LIN {X 0,Y 263.736,Z 330.131,A -85,B 0,C 180,E1 -17998.473,E2 -17998.473} C_VEL
LIN {X 0,Y 263.74,Z 330.122,A -85,B 0,C 180,E1 -18001.527,E2 -18001.527} C_VEL
LIN {X 0,Y 263.538,Z 330.145,A -85,B 0,C 180,E1 -18007.662,E2 -18007.662} C_VEL
LIN {X 0,Y 263.345,Z 330.181,A -85,B 0,C 180,E1 -18010.766,E2 -18010.766} C_VEL
LIN {X 0,Y 263.289,Z 330.157,A -85,B 0,C 180,E1 -18015.481,E2 -18015.481} C_VEL
LIN {X 0,Y 263.209,Z 330.198,A -85,B 0,C 180,E1 -18020.311,E2 -18020.311} C_VEL
LIN {X 0,Y 263.167,Z 330.188,A -85,B 0,C 180,E1 -18025.295,E2 -18025.295} C_VEL
LIN {X 0,Y 263.133,Z 330.206,A -85,B 0,C 180,E1 -18028.735,E2 -18028.735} C_VEL
LIN {X 0,Y 263.128,Z 330.196,A -85,B 0,C 180,E1 -18032.288,E2 -18032.288} C_VEL
LIN {X 0,Y 263.153,Z 330.198,A -85,B 0,C 180,E1 -18035.983,E2 -18035.983} C_VEL
LIN {X 0,Y 263.071,Z 330.217,A -85,B 0,C 180,E1 -18039.878,E2 -18039.878} C_VEL
LIN {X 0,Y 263.075,Z 330.212,A -85,B 0,C 180,E1 -18043.993,E2 -18043.993} C_VEL
LIN {X 0,Y 263.079,Z 330.215,A -85,B 0,C 180,E1 -18048.417,E2 -18048.417} C_VEL
LIN {X 0,Y 263.155,Z 330.203,A -85,B 0,C 180,E1 -18052.102,E2 -18052.102} C_VEL
LIN {X 0,Y 263.202,Z 330.409,A -85,B 0,C 180,E1 -18055.314,E2 -18055.314} C_VEL
LIN {X 0,Y 265.444,Z 340.558,A -85,B 0,C 180,E1 -18059.358,E2 -18059.358} C_VEL
LIN {X 0,Y 266.018,Z 343.587,A -85,B 0,C 180,E1 -18060.39,E2 -18060.39} C_VEL
LIN {X 0,Y 270.223,Z 354.313,A -85,B 0,C 180,E1 -18061.21,E2 -18061.21} C_VEL
LIN {X 0,Y 273.348,Z 362.999,A -85,B 0,C 180,E1 -18061.777,E2 -18061.777} C_VEL
LIN {X 0,Y 277.181,Z 387.27,A -85,B 0,C 180,E1 -18062.845,E2 -18062.845} C_VEL
LIN {X 0,Y 275.215,Z 449.746,A -85,B 0,C 180,E1 -18064.524,E2 -18064.524} C_VEL
LIN {X 0,Y 274.623,Z 459.446,A -85,B 0,C 180,E1 -18064.921,E2 -18064.921} C_VEL
LIN {X 0,Y 273.731,Z 469.978,A -85,B 0,C 180,E1 -18065.543,E2 -18065.543} C_VEL
LIN {X 0,Y 272.657,Z 479.225,A -85,B 0,C 180,E1 -18066.25,E2 -18066.25} C_VEL
LIN {X 0,Y 271.281,Z 490.013,A -85,B 0,C 180,E1 -18067.334,E2 -18067.334} C_VEL
LIN {X 0,Y 269.73,Z 500.089,A -85,B 0,C 180,E1 -18068.606,E2 -18068.606} C_VEL
LIN {X 0,Y 268.138,Z 509.514,A -85,B 0,C 180,E1 -18070.078,E2 -18070.078} C_VEL
LIN {X 0,Y 266.815,Z 517.421,A -85,B 0,C 180,E1 -18071.573,E2 -18071.573} C_VEL
LIN {X 0,Y 265.298,Z 525.618,A -85,B 0,C 180,E1 -18073.454,E2 -18073.454} C_VEL
LIN {X 0,Y 264.028,Z 532.435,A -85,B 0,C 180,E1 -18075.352,E2 -18075.352} C_VEL
LIN {X 0,Y 263.156,Z 537.135,A -85,B 0,C 180,E1 -18076.879,E2 -18076.879} C_VEL
LIN {X 0,Y 262.228,Z 542.864,A -85,B 0,C 180,E1 -18079.187,E2 -18079.187} C_VEL
LIN {X 0,Y 261.569,Z 547.363,A -85,B 0,C 180,E1 -18081.502,E2 -18081.502} C_VEL
LIN {X 0,Y 261.166,Z 550.77,A -85,B 0,C 180,E1 -18083.821,E2 -18083.821} C_VEL
LIN {X 0,Y 261.007,Z 553.667,A -85,B 0,C 180,E1 -18086.913,E2 -18086.913} C_VEL
LIN {X 0,Y 261.032,Z 554.618,A -85,B 0,C 180,E1 -18088.457,E2 -18088.457} C_VEL
LIN {X 0,Y 261.033,Z 555.058,A -85,B 0,C 180,E1 -18091.543,E2 -18091.543} C_VEL
LIN {X 0,Y 261.013,Z 554.722,A -85,B 0,C 180,E1 -18093.087,E2 -18093.087} C_VEL
LIN {X 0,Y 261.231,Z 552.837,A -85,B 0,C 180,E1 -18096.178,E2 -18096.178} C_VEL
LIN {X 0,Y 261.634,Z 550.327,A -85,B 0,C 180,E1 -18098.496,E2 -18098.496} C_VEL
LIN {X 0,Y 262.351,Z 546.813,A -85,B 0,C 180,E1 -18100.808,E2 -18100.808} C_VEL
LIN {X 0,Y 263.39,Z 542.211,A -85,B 0,C 180,E1 -18103.109,E2 -18103.109} C_VEL
LIN {X 0,Y 264.878,Z 536.377,A -85,B 0,C 180,E1 -18105.386,E2 -18105.386} C_VEL
LIN {X 0,Y 266.728,Z 529.069,A -85,B 0,C 180,E1 -18107.639,E2 -18107.639} C_VEL
LIN {X 0,Y 268.25,Z 522.147,A -85,B 0,C 180,E1 -18109.409,E2 -18109.409} C_VEL
LIN {X 0,Y 270.195,Z 513.761,A -85,B 0,C 180,E1 -18111.155,E2 -18111.155} C_VEL
LIN {X 0,Y 272.29,Z 504.136,A -85,B 0,C 180,E1 -18112.778,E2 -18112.778} C_VEL
LIN {X 0,Y 274.149,Z 495.111,A -85,B 0,C 180,E1 -18114.014,E2 -18114.014} C_VEL
LIN {X 0,Y 275.782,Z 485.768,A -85,B 0,C 180,E1 -18115.066,E2 -18115.066} C_VEL
LIN {X 0,Y 277.322,Z 475.015,A -85,B 0,C 180,E1 -18116.023,E2 -18116.023} C_VEL
LIN {X 0,Y 278.606,Z 464.155,A -85,B 0,C 180,E1 -18116.751,E2 -18116.751} C_VEL
LIN {X 0,Y 279.679,Z 453.063,A -85,B 0,C 180,E1 -18117.266,E2 -18117.266} C_VEL
LIN {X 0,Y 280.37,Z 435.148,A -85,B 0,C 180,E1 -18117.818,E2 -18117.818} C_VEL
LIN {X 0,Y 282.056,Z 388.472,A -85,B 0,C 180,E1 -18119.049,E2 -18119.049} C_VEL
LIN {X 0,Y 279.053,Z 370.079,A -85,B 0,C 180,E1 -18120.029,E2 -18120.029} C_VEL
LIN {X 0,Y 272.265,Z 354.512,A -85,B 0,C 180,E1 -18121.501,E2 -18121.501} C_VEL
LIN {X 0,Y 267.461,Z 345.107,A -85,B 0,C 180,E1 -18122.57,E2 -18122.57} C_VEL
LIN {X 0,Y 266.322,Z 342.4,A -85,B 0,C 180,E1 -18122.941,E2 -18122.941} C_VEL
LIN {X 0,Y 264.141,Z 333.763,A -85,B 0,C 180,E1 -18126.565,E2 -18126.565} C_VEL
LIN {X 0,Y 263.175,Z 330.249,A -85,B 0,C 180,E1 -18128.281,E2 -18128.281} C_VEL
LIN {X 0,Y 263.122,Z 330.208,A -85,B 0,C 180,E1 -18131.894,E2 -18131.894} C_VEL
LIN {X 0,Y 263.103,Z 330.208,A -85,B 0,C 180,E1 -18136.155,E2 -18136.155} C_VEL
LIN {X 0,Y 263.104,Z 330.212,A -85,B 0,C 180,E1 -18140.128,E2 -18140.128} C_VEL
LIN {X 0,Y 263.161,Z 330.2,A -85,B 0,C 180,E1 -18144.018,E2 -18144.018} C_VEL
LIN {X 0,Y 263.132,Z 330.203,A -85,B 0,C 180,E1 -18147.712,E2 -18147.712} C_VEL
LIN {X 0,Y 263.198,Z 330.194,A -85,B 0,C 180,E1 -18151.785,E2 -18151.785} C_VEL
LIN {X 0,Y 263.226,Z 330.195,A -85,B 0,C 180,E1 -18155.201,E2 -18155.201} C_VEL
LIN {X 0,Y 263.264,Z 330.19,A -85,B 0,C 180,E1 -18159.694,E2 -18159.694} C_VEL
LIN {X 0,Y 263.351,Z 330.179,A -85,B 0,C 180,E1 -18164.522,E2 -18164.522} C_VEL
LIN {X 0,Y 263.375,Z 330.178,A -85,B 0,C 180,E1 -18169.235,E2 -18169.235} C_VEL
LIN {X 0,Y 263.575,Z 330.146,A -85,B 0,C 180,E1 -18172.339,E2 -18172.339} C_VEL
LIN {X 0,Y 263.753,Z 330.131,A -85,B 0,C 180,E1 -18178.473,E2 -18178.473} C_VEL
LIN {X 0,Y 263.753,Z 330.125,A -85,B 0,C 180,E1 -18181.527,E2 -18181.527} C_VEL
LIN {X 0,Y 263.574,Z 330.15,A -85,B 0,C 180,E1 -18187.662,E2 -18187.662} C_VEL
LIN {X 0,Y 263.376,Z 330.178,A -85,B 0,C 180,E1 -18190.766,E2 -18190.766} C_VEL
LIN {X 0,Y 263.352,Z 330.176,A -85,B 0,C 180,E1 -18195.478,E2 -18195.478} C_VEL
LIN {X 0,Y 263.263,Z 330.192,A -85,B 0,C 180,E1 -18200.307,E2 -18200.307} C_VEL
LIN {X 0,Y 263.186,Z 330.202,A -85,B 0,C 180,E1 -18205.294,E2 -18205.294} C_VEL
LIN {X 0,Y 263.164,Z 330.203,A -85,B 0,C 180,E1 -18209.828,E2 -18209.828} C_VEL
LIN {X 0,Y 263.23,Z 330.519,A -85,B 0,C 180,E1 -18210.262,E2 -18210.262} C_VEL
LIN {X 0,Y 264.944,Z 336.603,A -85,B 0,C 180,E1 -18212.886,E2 -18212.886} C_VEL
LIN {X 0,Y 267.825,Z 342.072,A -85,B 0,C 180,E1 -18213.63,E2 -18213.63} C_VEL
LIN {X 0,Y 274.766,Z 355.657,A -85,B 0,C 180,E1 -18215.15,E2 -18215.15} C_VEL
LIN {X 0,Y 281.344,Z 371.108,A -85,B 0,C 180,E1 -18216.558,E2 -18216.558} C_VEL
LIN {X 0,Y 282.522,Z 377.532,A -85,B 0,C 180,E1 -18216.915,E2 -18216.915} C_VEL
LIN {X 0,Y 279.879,Z 443.081,A -85,B 0,C 180,E1 -18218.66,E2 -18218.66} C_VEL
LIN {X 0,Y 279.168,Z 453.092,A -85,B 0,C 180,E1 -18219.075,E2 -18219.075} C_VEL
LIN {X 0,Y 278.267,Z 462.472,A -85,B 0,C 180,E1 -18219.618,E2 -18219.618} C_VEL
LIN {X 0,Y 276.999,Z 472.966,A -85,B 0,C 180,E1 -18220.434,E2 -18220.434} C_VEL
LIN {X 0,Y 275.434,Z 482.994,A -85,B 0,C 180,E1 -18221.423,E2 -18221.423} C_VEL
LIN {X 0,Y 273.661,Z 493.048,A -85,B 0,C 180,E1 -18222.682,E2 -18222.682} C_VEL
LIN {X 0,Y 271.796,Z 502.27,A -85,B 0,C 180,E1 -18224.104,E2 -18224.104} C_VEL
LIN {X 0,Y 269.717,Z 511.296,A -85,B 0,C 180,E1 -18225.812,E2 -18225.812} C_VEL
LIN {X 0,Y 267.874,Z 518.886,A -85,B 0,C 180,E1 -18227.565,E2 -18227.565} C_VEL
LIN {X 0,Y 266.451,Z 524.682,A -85,B 0,C 180,E1 -18229.155,E2 -18229.155} C_VEL
LIN {X 0,Y 264.768,Z 531.329,A -85,B 0,C 180,E1 -18231.407,E2 -18231.407} C_VEL
LIN {X 0,Y 263.723,Z 535.462,A -85,B 0,C 180,E1 -18233.08,E2 -18233.08} C_VEL
LIN {X 0,Y 262.444,Z 540.564,A -85,B 0,C 180,E1 -18235.781,E2 -18235.781} C_VEL
LIN {X 0,Y 261.865,Z 543.167,A -85,B 0,C 180,E1 -18237.536,E2 -18237.536} C_VEL
LIN {X 0,Y 261.377,Z 545.131,A -85,B 0,C 180,E1 -18239.365,E2 -18239.365} C_VEL
LIN {X 0,Y 260.81,Z 547.438,A -85,B 0,C 180,E1 -18242.736,E2 -18242.736} C_VEL
LIN {X 0,Y 260.66,Z 547.783,A -85,B 0,C 180,E1 -18244.444,E2 -18244.444} C_VEL
LIN {X 0,Y 260.664,Z 547.185,A -85,B 0,C 180,E1 -18247.823,E2 -18247.823} C_VEL
LIN {X 0,Y 260.965,Z 545.286,A -85,B 0,C 180,E1 -18250.49,E2 -18250.49} C_VEL
LIN {X 0,Y 261.376,Z 542.668,A -85,B 0,C 180,E1 -18252.796,E2 -18252.796} C_VEL
LIN {X 0,Y 261.913,Z 539.194,A -85,B 0,C 180,E1 -18255.017,E2 -18255.017} C_VEL
LIN {X 0,Y 262.505,Z 535.554,A -85,B 0,C 180,E1 -18256.846,E2 -18256.846} C_VEL
LIN {X 0,Y 263.528,Z 529.579,A -85,B 0,C 180,E1 -18259.241,E2 -18259.241} C_VEL
LIN {X 0,Y 264.959,Z 521.962,A -85,B 0,C 180,E1 -18261.612,E2 -18261.612} C_VEL
LIN {X 0,Y 266.44,Z 514.196,A -85,B 0,C 180,E1 -18263.564,E2 -18263.564} C_VEL
LIN {X 0,Y 267.763,Z 506.654,A -85,B 0,C 180,E1 -18265.145,E2 -18265.145} C_VEL
LIN {X 0,Y 269.281,Z 498.066,A -85,B 0,C 180,E1 -18266.634,E2 -18266.634} C_VEL
LIN {X 0,Y 270.742,Z 488.817,A -85,B 0,C 180,E1 -18267.955,E2 -18267.955} C_VEL
LIN {X 0,Y 272.075,Z 479.203,A -85,B 0,C 180,E1 -18269.075,E2 -18269.075} C_VEL
LIN {X 0,Y 273.277,Z 469.269,A -85,B 0,C 180,E1 -18270,E2 -18270} C_VEL
LIN {X 0,Y 274.319,Z 457.387,A -85,B 0,C 180,E1 -18270.836,E2 -18270.836} C_VEL
LIN {X 0,Y 275.192,Z 445.994,A -85,B 0,C 180,E1 -18271.385,E2 -18271.385} C_VEL
LIN {X 0,Y 275.864,Z 428.906,A -85,B 0,C 180,E1 -18271.899,E2 -18271.899} C_VEL
LIN {X 0,Y 277.459,Z 374.822,A -85,B 0,C 180,E1 -18273.325,E2 -18273.325} C_VEL
LIN {X 0,Y 275.15,Z 362.729,A -85,B 0,C 180,E1 -18273.899,E2 -18273.899} C_VEL
LIN {X 0,Y 269.038,Z 346.952,A -85,B 0,C 180,E1 -18274.974,E2 -18274.974} C_VEL
LIN {X 0,Y 264.977,Z 337.261,A -85,B 0,C 180,E1 -18275.747,E2 -18275.747} C_VEL
LIN {X 0,Y 264.714,Z 335.941,A -85,B 0,C 180,E1 -18276.096,E2 -18276.096} C_VEL
LIN {X 0,Y 263.505,Z 330.211,A -85,B 0,C 180,E1 -18278.548,E2 -18278.548} C_VEL
LIN {X 0,Y 263.324,Z 330.174,A -85,B 0,C 180,E1 -18282.329,E2 -18282.329} C_VEL
LIN {X 0,Y 263.349,Z 330.177,A -85,B 0,C 180,E1 -18286.109,E2 -18286.109} C_VEL
LIN {X 0,Y 263.216,Z 330.199,A -85,B 0,C 180,E1 -18290.849,E2 -18290.849} C_VEL
LIN {X 0,Y 263.195,Z 330.201,A -85,B 0,C 180,E1 -18295.293,E2 -18295.293} C_VEL
LIN {X 0,Y 263.168,Z 330.189,A -85,B 0,C 180,E1 -18298.731,E2 -18298.731} C_VEL
LIN {X 0,Y 263.135,Z 330.204,A -85,B 0,C 180,E1 -18302.288,E2 -18302.288} C_VEL
LIN {X 0,Y 263.189,Z 330.191,A -85,B 0,C 180,E1 -18305.978,E2 -18305.978} C_VEL
LIN {X 0,Y 263.117,Z 330.198,A -85,B 0,C 180,E1 -18309.871,E2 -18309.871} C_VEL
LIN {X 0,Y 263.13,Z 330.199,A -85,B 0,C 180,E1 -18313.983,E2 -18313.983} C_VEL
LIN {X 0,Y 263.127,Z 330.193,A -85,B 0,C 180,E1 -18318.406,E2 -18318.406} C_VEL
LIN {X 0,Y 263.16,Z 330.185,A -85,B 0,C 180,E1 -18322.103,E2 -18322.103} C_VEL
LIN {X 0,Y 263.153,Z 330.202,A -85,B 0,C 180,E1 -18325.885,E2 -18325.885} C_VEL
LIN {X 0,Y 263.128,Z 330.174,A -85,B 0,C 180,E1 -18329.504,E2 -18329.504} C_VEL
LIN {X 0,Y 263.151,Z 330.19,A -85,B 0,C 180,E1 -18332.998,E2 -18332.998} C_VEL
LIN {X 0,Y 263.152,Z 330.206,A -85,B 0,C 180,E1 -18336.384,E2 -18336.384} C_VEL
LIN {X 0,Y 263.24,Z 330.172,A -85,B 0,C 180,E1 -18339.691,E2 -18339.691} C_VEL
LIN {X 0,Y 263.317,Z 330.165,A -85,B 0,C 180,E1 -18344.52,E2 -18344.52} C_VEL
LIN {X 0,Y 263.355,Z 330.176,A -85,B 0,C 180,E1 -18349.233,E2 -18349.233} C_VEL
LIN {X 0,Y 263.528,Z 330.124,A -85,B 0,C 180,E1 -18352.337,E2 -18352.337} C_VEL
LIN {X 0,Y 263.478,Z 330.122,A -85,B 0,C 180,E1 -18353.306,E2 -18353.306} C_VEL
LIN {X 0,Y 262.843,Z 330.206,A -85,B 0,C 180,E1 -18354.581,E2 -18354.581} C_VEL
LIN {X 0,Y 260.134,Z 330.568,A -85,B 0,C 180,E1 -18356.665,E2 -18356.665} C_VEL
LIN {X 0,Y 257.028,Z 330.971,A -85,B 0,C 180,E1 -18359.227,E2 -18359.227} C_VEL
LIN {X 0,Y 256.696,Z 331.007,A -85,B 0,C 180,E1 -18360.112,E2 -18360.112} C_VEL
LIN {X 0,Y 256.702,Z 330.999,A -85,B 0,C 180,E1 -18361.568,E2 -18361.568} C_VEL
LIN {X 0,Y 256.464,Z 331.01,A -85,B 0,C 180,E1 -18366.293,E2 -18366.293} C_VEL
LIN {X 0,Y 256.428,Z 331.044,A -85,B 0,C 180,E1 -18369.464,E2 -18369.464} C_VEL
LIN {X 0,Y 256.207,Z 331.04,A -85,B 0,C 180,E1 -18374.292,E2 -18374.292} C_VEL
LIN {X 0,Y 256.149,Z 331.066,A -85,B 0,C 180,E1 -18377.566,E2 -18377.566} C_VEL
LIN {X 0,Y 256.122,Z 331.076,A -85,B 0,C 180,E1 -18381.098,E2 -18381.098} C_VEL
LIN {X 0,Y 256.133,Z 331.061,A -85,B 0,C 180,E1 -18385.111,E2 -18385.111} C_VEL
LIN {X 0,Y 256.055,Z 331.08,A -85,B 0,C 180,E1 -18389.607,E2 -18389.607} C_VEL
LIN {X 0,Y 256.066,Z 331.083,A -85,B 0,C 180,E1 -18393.292,E2 -18393.292} C_VEL
LIN {X 0,Y 256.086,Z 331.072,A -85,B 0,C 180,E1 -18397.262,E2 -18397.262} C_VEL
LIN {X 0,Y 256.007,Z 331.092,A -85,B 0,C 180,E1 -18401.212,E2 -18401.212} C_VEL
LIN {X 0,Y 256.016,Z 331.092,A -85,B 0,C 180,E1 -18405.539,E2 -18405.539} C_VEL
LIN {X 0,Y 256.016,Z 331.092,A -85,B 0,C 180,E1 -18408.789,E2 -18408.789} C_VEL
LIN {X 0,Y 256.124,Z 331.084,A -85,B 0,C 180,E1 -18412.866,E2 -18412.866} C_VEL
LIN {X 0,Y 256.132,Z 331.241,A -85,B 0,C 180,E1 -18414.694,E2 -18414.694} C_VEL
LIN {X 0,Y 258.047,Z 339.906,A -85,B 0,C 180,E1 -18418.295,E2 -18418.295} C_VEL
LIN {X 0,Y 258.824,Z 343.419,A -85,B 0,C 180,E1 -18419.59,E2 -18419.59} C_VEL
LIN {X 0,Y 262.014,Z 351.634,A -85,B 0,C 180,E1 -18420.266,E2 -18420.266} C_VEL
LIN {X 0,Y 267.097,Z 365.128,A -85,B 0,C 180,E1 -18421.216,E2 -18421.216} C_VEL
LIN {X 0,Y 270.669,Z 388.523,A -85,B 0,C 180,E1 -18422.271,E2 -18422.271} C_VEL
LIN {X 0,Y 268.653,Z 449.918,A -85,B 0,C 180,E1 -18423.96,E2 -18423.96} C_VEL
LIN {X 0,Y 268.052,Z 459.524,A -85,B 0,C 180,E1 -18424.366,E2 -18424.366} C_VEL
LIN {X 0,Y 267.133,Z 470.01,A -85,B 0,C 180,E1 -18425.002,E2 -18425.002} C_VEL
LIN {X 0,Y 265.912,Z 480.168,A -85,B 0,C 180,E1 -18425.816,E2 -18425.816} C_VEL
LIN {X 0,Y 264.461,Z 490.751,A -85,B 0,C 180,E1 -18426.922,E2 -18426.922} C_VEL
LIN {X 0,Y 262.882,Z 500.682,A -85,B 0,C 180,E1 -18428.226,E2 -18428.226} C_VEL
LIN {X 0,Y 261.399,Z 508.961,A -85,B 0,C 180,E1 -18429.542,E2 -18429.542} C_VEL
LIN {X 0,Y 260.072,Z 516.951,A -85,B 0,C 180,E1 -18431.078,E2 -18431.078} C_VEL
LIN {X 0,Y 258.474,Z 525.213,A -85,B 0,C 180,E1 -18433.004,E2 -18433.004} C_VEL
LIN {X 0,Y 257.133,Z 532.085,A -85,B 0,C 180,E1 -18434.95,E2 -18434.95} C_VEL
LIN {X 0,Y 256.214,Z 536.809,A -85,B 0,C 180,E1 -18436.517,E2 -18436.517} C_VEL
LIN {X 0,Y 255.209,Z 542.597,A -85,B 0,C 180,E1 -18438.885,E2 -18438.885} C_VEL
LIN {X 0,Y 254.542,Z 547.14,A -85,B 0,C 180,E1 -18441.265,E2 -18441.265} C_VEL
LIN {X 0,Y 254.082,Z 550.579,A -85,B 0,C 180,E1 -18443.648,E2 -18443.648} C_VEL
LIN {X 0,Y 253.911,Z 553.518,A -85,B 0,C 180,E1 -18446.826,E2 -18446.826} C_VEL
LIN {X 0,Y 253.942,Z 554.478,A -85,B 0,C 180,E1 -18448.414,E2 -18448.414} C_VEL
LIN {X 0,Y 253.942,Z 554.974,A -85,B 0,C 180,E1 -18451.586,E2 -18451.586} C_VEL
LIN {X 0,Y 253.916,Z 554.639,A -85,B 0,C 180,E1 -18453.173,E2 -18453.173} C_VEL
LIN {X 0,Y 254.162,Z 552.82,A -85,B 0,C 180,E1 -18456.35,E2 -18456.35} C_VEL
LIN {X 0,Y 254.828,Z 549.202,A -85,B 0,C 180,E1 -18459.525,E2 -18459.525} C_VEL
LIN {X 0,Y 255.698,Z 545.374,A -85,B 0,C 180,E1 -18461.896,E2 -18461.896} C_VEL
LIN {X 0,Y 256.462,Z 542.3,A -85,B 0,C 180,E1 -18463.47,E2 -18463.47} C_VEL
LIN {X 0,Y 258.383,Z 535.357,A -85,B 0,C 180,E1 -18466.188,E2 -18466.188} C_VEL
LIN {X 0,Y 259.963,Z 529.277,A -85,B 0,C 180,E1 -18468.113,E2 -18468.113} C_VEL
LIN {X 0,Y 261.749,Z 521.63,A -85,B 0,C 180,E1 -18470.1,E2 -18470.1} C_VEL
LIN {X 0,Y 263.861,Z 513.091,A -85,B 0,C 180,E1 -18471.894,E2 -18471.894} C_VEL
LIN {X 0,Y 265.771,Z 504.595,A -85,B 0,C 180,E1 -18473.369,E2 -18473.369} C_VEL
LIN {X 0,Y 267.717,Z 495.707,A -85,B 0,C 180,E1 -18474.629,E2 -18474.629} C_VEL
LIN {X 0,Y 269.4,Z 486.556,A -85,B 0,C 180,E1 -18475.703,E2 -18475.703} C_VEL
LIN {X 0,Y 271.18,Z 474.889,A -85,B 0,C 180,E1 -18476.763,E2 -18476.763} C_VEL
LIN {X 0,Y 272.492,Z 464.05,A -85,B 0,C 180,E1 -18477.505,E2 -18477.505} C_VEL
LIN {X 0,Y 273.602,Z 452.945,A -85,B 0,C 180,E1 -18478.029,E2 -18478.029} C_VEL
LIN {X 0,Y 274.368,Z 434.186,A -85,B 0,C 180,E1 -18478.613,E2 -18478.613} C_VEL
LIN {X 0,Y 276.065,Z 389.46,A -85,B 0,C 180,E1 -18479.816,E2 -18479.816} C_VEL
LIN {X 0,Y 273.349,Z 372.72,A -85,B 0,C 180,E1 -18480.74,E2 -18480.74} C_VEL
LIN {X 0,Y 267.024,Z 358.117,A -85,B 0,C 180,E1 -18482.185,E2 -18482.185} C_VEL
LIN {X 0,Y 260.612,Z 345.455,A -85,B 0,C 180,E1 -18483.695,E2 -18483.695} C_VEL
LIN {X 0,Y 259.105,Z 342.293,A -85,B 0,C 180,E1 -18484.148,E2 -18484.148} C_VEL
LIN {X 0,Y 257.049,Z 334.623,A -85,B 0,C 180,E1 -18487.544,E2 -18487.544} C_VEL
LIN {X 0,Y 256.096,Z 331.129,A -85,B 0,C 180,E1 -18489.336,E2 -18489.336} C_VEL
LIN {X 0,Y 256.047,Z 331.088,A -85,B 0,C 180,E1 -18493.33,E2 -18493.33} C_VEL
LIN {X 0,Y 256.068,Z 331.084,A -85,B 0,C 180,E1 -18497.82,E2 -18497.82} C_VEL
LIN {X 0,Y 256.07,Z 331.084,A -85,B 0,C 180,E1 -18500.858,E2 -18500.858} C_VEL
LIN {X 0,Y 256.129,Z 331.081,A -85,B 0,C 180,E1 -18502.868,E2 -18502.868} C_VEL
LIN {X 0,Y 256.067,Z 331.089,A -85,B 0,C 180,E1 -18506.708,E2 -18506.708} C_VEL
LIN {X 0,Y 256.11,Z 331.084,A -85,B 0,C 180,E1 -18510.4,E2 -18510.4} C_VEL
LIN {X 0,Y 256.188,Z 331.074,A -85,B 0,C 180,E1 -18514.862,E2 -18514.862} C_VEL
LIN {X 0,Y 256.167,Z 331.077,A -85,B 0,C 180,E1 -18519.105,E2 -18519.105} C_VEL
LIN {X 0,Y 256.301,Z 331.058,A -85,B 0,C 180,E1 -18524.086,E2 -18524.086} C_VEL
LIN {X 0,Y 256.311,Z 331.057,A -85,B 0,C 180,E1 -18528.934,E2 -18528.934} C_VEL
LIN {X 0,Y 256.542,Z 331.02,A -85,B 0,C 180,E1 -18532.128,E2 -18532.128} C_VEL
LIN {X 0,Y 256.716,Z 331.008,A -85,B 0,C 180,E1 -18538.432,E2 -18538.432} C_VEL
LIN {X 0,Y 256.716,Z 331.002,A -85,B 0,C 180,E1 -18541.569,E2 -18541.569} C_VEL
LIN {X 0,Y 256.542,Z 331.025,A -85,B 0,C 180,E1 -18547.873,E2 -18547.873} C_VEL
LIN {X 0,Y 256.311,Z 331.06,A -85,B 0,C 180,E1 -18551.066,E2 -18551.066} C_VEL
LIN {X 0,Y 256.301,Z 331.053,A -85,B 0,C 180,E1 -18555.915,E2 -18555.915} C_VEL
LIN {X 0,Y 256.163,Z 331.077,A -85,B 0,C 180,E1 -18560.896,E2 -18560.896} C_VEL
LIN {X 0,Y 256.167,Z 331.075,A -85,B 0,C 180,E1 -18565.128,E2 -18565.128} C_VEL
LIN {X 0,Y 256.156,Z 331.242,A -85,B 0,C 180,E1 -18569.115,E2 -18569.115} C_VEL
LIN {X 0,Y 257.732,Z 336.832,A -85,B 0,C 180,E1 -18571.672,E2 -18571.672} C_VEL
LIN {X 0,Y 264.661,Z 349.466,A -85,B 0,C 180,E1 -18573.38,E2 -18573.38} C_VEL
LIN {X 0,Y 271.508,Z 363.737,A -85,B 0,C 180,E1 -18574.94,E2 -18574.94} C_VEL
LIN {X 0,Y 275.907,Z 374.539,A -85,B 0,C 180,E1 -18575.926,E2 -18575.926} C_VEL
LIN {X 0,Y 276.545,Z 379.133,A -85,B 0,C 180,E1 -18576.163,E2 -18576.163} C_VEL
LIN {X 0,Y 273.894,Z 442.189,A -85,B 0,C 180,E1 -18577.865,E2 -18577.865} C_VEL
LIN {X 0,Y 273.133,Z 452.692,A -85,B 0,C 180,E1 -18578.293,E2 -18578.293} C_VEL
LIN {X 0,Y 272.01,Z 463.583,A -85,B 0,C 180,E1 -18578.946,E2 -18578.946} C_VEL
LIN {X 0,Y 270.751,Z 473.437,A -85,B 0,C 180,E1 -18579.737,E2 -18579.737} C_VEL
LIN {X 0,Y 269.091,Z 483.537,A -85,B 0,C 180,E1 -18580.764,E2 -18580.764} C_VEL
LIN {X 0,Y 267.269,Z 493.352,A -85,B 0,C 180,E1 -18582.025,E2 -18582.025} C_VEL
LIN {X 0,Y 265.224,Z 502.922,A -85,B 0,C 180,E1 -18583.548,E2 -18583.548} C_VEL
LIN {X 0,Y 263.411,Z 510.538,A -85,B 0,C 180,E1 -18585.006,E2 -18585.006} C_VEL
LIN {X 0,Y 261.374,Z 518.518,A -85,B 0,C 180,E1 -18586.864,E2 -18586.864} C_VEL
LIN {X 0,Y 259.469,Z 525.768,A -85,B 0,C 180,E1 -18588.941,E2 -18588.941} C_VEL
LIN {X 0,Y 258.126,Z 530.959,A -85,B 0,C 180,E1 -18590.733,E2 -18590.733} C_VEL
LIN {X 0,Y 256.683,Z 536.199,A -85,B 0,C 180,E1 -18592.961,E2 -18592.961} C_VEL
LIN {X 0,Y 255.809,Z 539.652,A -85,B 0,C 180,E1 -18594.764,E2 -18594.764} C_VEL
LIN {X 0,Y 254.79,Z 543.575,A -85,B 0,C 180,E1 -18597.461,E2 -18597.461} C_VEL
LIN {X 0,Y 254.096,Z 546.171,A -85,B 0,C 180,E1 -18600.142,E2 -18600.142} C_VEL
LIN {X 0,Y 253.752,Z 547.494,A -85,B 0,C 180,E1 -18602.41,E2 -18602.41} C_VEL
LIN {X 0,Y 253.53,Z 547.9,A -85,B 0,C 180,E1 -18605.43,E2 -18605.43} C_VEL
LIN {X 0,Y 253.554,Z 547.536,A -85,B 0,C 180,E1 -18607.167,E2 -18607.167} C_VEL
LIN {X 0,Y 253.885,Z 545.315,A -85,B 0,C 180,E1 -18610.599,E2 -18610.599} C_VEL
LIN {X 0,Y 254.354,Z 542.424,A -85,B 0,C 180,E1 -18613.135,E2 -18613.135} C_VEL
LIN {X 0,Y 254.782,Z 539.814,A -85,B 0,C 180,E1 -18614.897,E2 -18614.897} C_VEL
LIN {X 0,Y 255.55,Z 535.17,A -85,B 0,C 180,E1 -18617.29,E2 -18617.29} C_VEL
LIN {X 0,Y 256.855,Z 528.022,A -85,B 0,C 180,E1 -18620.073,E2 -18620.073} C_VEL
LIN {X 0,Y 257.934,Z 522.704,A -85,B 0,C 180,E1 -18621.776,E2 -18621.776} C_VEL
LIN {X 0,Y 259.433,Z 515.067,A -85,B 0,C 180,E1 -18623.779,E2 -18623.779} C_VEL
LIN {X 0,Y 261.066,Z 506.209,A -85,B 0,C 180,E1 -18625.672,E2 -18625.672} C_VEL
LIN {X 0,Y 262.571,Z 497.979,A -85,B 0,C 180,E1 -18627.123,E2 -18627.123} C_VEL
LIN {X 0,Y 264.056,Z 488.705,A -85,B 0,C 180,E1 -18628.475,E2 -18628.475} C_VEL
LIN {X 0,Y 265.461,Z 479.018,A -85,B 0,C 180,E1 -18629.621,E2 -18629.621} C_VEL
LIN {X 0,Y 266.784,Z 468.236,A -85,B 0,C 180,E1 -18630.624,E2 -18630.624} C_VEL
LIN {X 0,Y 267.795,Z 456.72,A -85,B 0,C 180,E1 -18631.435,E2 -18631.435} C_VEL
LIN {X 0,Y 268.665,Z 445.602,A -85,B 0,C 180,E1 -18631.971,E2 -18631.971} C_VEL
LIN {X 0,Y 269.365,Z 427.888,A -85,B 0,C 180,E1 -18632.51,E2 -18632.51} C_VEL
LIN {X 0,Y 271.02,Z 376.113,A -85,B 0,C 180,E1 -18633.899,E2 -18633.899} C_VEL
LIN {X 0,Y 268.953,Z 365.142,A -85,B 0,C 180,E1 -18634.434,E2 -18634.434} C_VEL
LIN {X 0,Y 263.196,Z 350.275,A -85,B 0,C 180,E1 -18635.483,E2 -18635.483} C_VEL
LIN {X 0,Y 257.83,Z 337.321,A -85,B 0,C 180,E1 -18636.53,E2 -18636.53} C_VEL
LIN {X 0,Y 257.473,Z 335.653,A -85,B 0,C 180,E1 -18637.056,E2 -18637.056} C_VEL
LIN {X 0,Y 256.45,Z 331.081,A -85,B 0,C 180,E1 -18639.131,E2 -18639.131} C_VEL
LIN {X 0,Y 256.257,Z 331.063,A -85,B 0,C 180,E1 -18644.29,E2 -18644.29} C_VEL
LIN {X 0,Y 256.212,Z 331.071,A -85,B 0,C 180,E1 -18647.562,E2 -18647.562} C_VEL
LIN {X 0,Y 256.156,Z 331.077,A -85,B 0,C 180,E1 -18651.118,E2 -18651.118} C_VEL
LIN {X 0,Y 256.173,Z 331.076,A -85,B 0,C 180,E1 -18655.13,E2 -18655.13} C_VEL
LIN {X 0,Y 256.106,Z 331.076,A -85,B 0,C 180,E1 -18659.601,E2 -18659.601} C_VEL
LIN {X 0,Y 256.087,Z 331.07,A -85,B 0,C 180,E1 -18663.29,E2 -18663.29} C_VEL
LIN {X 0,Y 256.13,Z 331.079,A -85,B 0,C 180,E1 -18667.275,E2 -18667.275} C_VEL
LIN {X 0,Y 256.059,Z 331.066,A -85,B 0,C 180,E1 -18671.203,E2 -18671.203} C_VEL
LIN {X 0,Y 256.064,Z 331.087,A -85,B 0,C 180,E1 -18675.529,E2 -18675.529} C_VEL
LIN {X 0,Y 256.056,Z 331.068,A -85,B 0,C 180,E1 -18678.797,E2 -18678.797} C_VEL
LIN {X 0,Y 256.13,Z 331.065,A -85,B 0,C 180,E1 -18682.867,E2 -18682.867} C_VEL
LIN {X 0,Y 256.068,Z 331.084,A -85,B 0,C 180,E1 -18686.707,E2 -18686.707} C_VEL
LIN {X 0,Y 256.057,Z 331.048,A -85,B 0,C 180,E1 -18690.393,E2 -18690.393} C_VEL
LIN {X 0,Y 256.163,Z 331.073,A -85,B 0,C 180,E1 -18694.875,E2 -18694.875} C_VEL
LIN {X 0,Y 256.151,Z 331.06,A -85,B 0,C 180,E1 -18699.103,E2 -18699.103} C_VEL
LIN {X 0,Y 256.251,Z 331.041,A -85,B 0,C 180,E1 -18704.082,E2 -18704.082} C_VEL
LIN {X 0,Y 256.291,Z 331.06,A -85,B 0,C 180,E1 -18707.327,E2 -18707.327} C_VEL
LIN {X 0,Y 256.436,Z 331.028,A -85,B 0,C 180,E1 -18710.622,E2 -18710.622} C_VEL
LIN {X 0,Y 256.457,Z 330.995,A -85,B 0,C 180,E1 -18713.706,E2 -18713.706} C_VEL
LIN {X 0,Y 256.698,Z 331.007,A -85,B 0,C 180,E1 -18718.431,E2 -18718.431} C_VEL
LIN {X 0,Y 256.696,Z 331.007,A -85,B 0,C 180,E1 -18720.112,E2 -18720.112} C_VEL
LIN {X 0,Y 255.97,Z 331.091,A -85,B 0,C 180,E1 -18721.417,E2 -18721.417} C_VEL
LIN {X 0,Y 253.034,Z 331.435,A -85,B 0,C 180,E1 -18723.543,E2 -18723.543} C_VEL
LIN {X 0,Y 250.564,Z 331.74,A -85,B 0,C 180,E1 -18725.273,E2 -18725.273} C_VEL
LIN {X 0,Y 249.504,Z 331.879,A -85,B 0,C 180,E1 -18726.617,E2 -18726.617} C_VEL
LIN {X 0,Y 249.416,Z 331.893,A -85,B 0,C 180,E1 -18727.073,E2 -18727.073} C_VEL
LIN {X 0,Y 249.343,Z 331.926,A -85,B 0,C 180,E1 -18729.736,E2 -18729.736} C_VEL
LIN {X 0,Y 249.15,Z 331.917,A -85,B 0,C 180,E1 -18734.706,E2 -18734.706} C_VEL
LIN {X 0,Y 249.081,Z 331.951,A -85,B 0,C 180,E1 -18738.081,E2 -18738.081} C_VEL
LIN {X 0,Y 249.046,Z 331.957,A -85,B 0,C 180,E1 -18741.521,E2 -18741.521} C_VEL
LIN {X 0,Y 249.085,Z 331.943,A -85,B 0,C 180,E1 -18745.459,E2 -18745.459} C_VEL
LIN {X 0,Y 249.037,Z 331.959,A -85,B 0,C 180,E1 -18748.973,E2 -18748.973} C_VEL
LIN {X 0,Y 249.027,Z 331.953,A -85,B 0,C 180,E1 -18752.426,E2 -18752.426} C_VEL
LIN {X 0,Y 249.01,Z 331.958,A -85,B 0,C 180,E1 -18756.348,E2 -18756.348} C_VEL
LIN {X 0,Y 248.97,Z 331.971,A -85,B 0,C 180,E1 -18760.484,E2 -18760.484} C_VEL
LIN {X 0,Y 248.961,Z 331.973,A -85,B 0,C 180,E1 -18764.888,E2 -18764.888} C_VEL
LIN {X 0,Y 248.991,Z 331.969,A -85,B 0,C 180,E1 -18767.357,E2 -18767.357} C_VEL
LIN {X 0,Y 249.039,Z 331.962,A -85,B 0,C 180,E1 -18772.201,E2 -18772.201} C_VEL
LIN {X 0,Y 249.091,Z 332.007,A -85,B 0,C 180,E1 -18774.005,E2 -18774.005} C_VEL
LIN {X 0,Y 250.44,Z 338.02,A -85,B 0,C 180,E1 -18776.66,E2 -18776.66} C_VEL
LIN {X 0,Y 251.549,Z 343.313,A -85,B 0,C 180,E1 -18778.739,E2 -18778.739} C_VEL
LIN {X 0,Y 255.964,Z 354.249,A -85,B 0,C 180,E1 -18779.674,E2 -18779.674} C_VEL
LIN {X 0,Y 260.933,Z 367.589,A -85,B 0,C 180,E1 -18780.645,E2 -18780.645} C_VEL
LIN {X 0,Y 264.204,Z 389.296,A -85,B 0,C 180,E1 -18781.658,E2 -18781.658} C_VEL
LIN {X 0,Y 262.122,Z 449.981,A -85,B 0,C 180,E1 -18783.367,E2 -18783.367} C_VEL
LIN {X 0,Y 261.506,Z 459.528,A -85,B 0,C 180,E1 -18783.784,E2 -18783.784} C_VEL
LIN {X 0,Y 260.535,Z 469.981,A -85,B 0,C 180,E1 -18784.43,E2 -18784.43} C_VEL
LIN {X 0,Y 259.408,Z 479.185,A -85,B 0,C 180,E1 -18785.169,E2 -18785.169} C_VEL
LIN {X 0,Y 257.913,Z 489.943,A -85,B 0,C 180,E1 -18786.301,E2 -18786.301} C_VEL
LIN {X 0,Y 256.228,Z 499.996,A -85,B 0,C 180,E1 -18787.631,E2 -18787.631} C_VEL
LIN {X 0,Y 254.513,Z 509.407,A -85,B 0,C 180,E1 -18789.174,E2 -18789.174} C_VEL
LIN {X 0,Y 253.18,Z 517.086,A -85,B 0,C 180,E1 -18790.699,E2 -18790.699} C_VEL
LIN {X 0,Y 251.674,Z 524.78,A -85,B 0,C 180,E1 -18792.531,E2 -18792.531} C_VEL
LIN {X 0,Y 250.262,Z 531.711,A -85,B 0,C 180,E1 -18794.527,E2 -18794.527} C_VEL
LIN {X 0,Y 248.847,Z 538.463,A -85,B 0,C 180,E1 -18796.942,E2 -18796.942} C_VEL
LIN {X 0,Y 248.209,Z 542.302,A -85,B 0,C 180,E1 -18798.568,E2 -18798.568} C_VEL
LIN {X 0,Y 247.506,Z 546.894,A -85,B 0,C 180,E1 -18801.015,E2 -18801.015} C_VEL
LIN {X 0,Y 247.025,Z 550.371,A -85,B 0,C 180,E1 -18803.465,E2 -18803.465} C_VEL
LIN {X 0,Y 246.818,Z 553.363,A -85,B 0,C 180,E1 -18806.735,E2 -18806.735} C_VEL
LIN {X 0,Y 246.853,Z 554.329,A -85,B 0,C 180,E1 -18808.368,E2 -18808.368} C_VEL
LIN {X 0,Y 246.854,Z 554.893,A -85,B 0,C 180,E1 -18811.631,E2 -18811.631} C_VEL
LIN {X 0,Y 246.823,Z 554.557,A -85,B 0,C 180,E1 -18813.264,E2 -18813.264} C_VEL
LIN {X 0,Y 247.081,Z 552.798,A -85,B 0,C 180,E1 -18816.533,E2 -18816.533} C_VEL
LIN {X 0,Y 247.817,Z 549.23,A -85,B 0,C 180,E1 -18819.797,E2 -18819.797} C_VEL
LIN {X 0,Y 248.727,Z 545.441,A -85,B 0,C 180,E1 -18822.235,E2 -18822.235} C_VEL
LIN {X 0,Y 249.977,Z 540.533,A -85,B 0,C 180,E1 -18824.657,E2 -18824.657} C_VEL
LIN {X 0,Y 251.562,Z 535.526,A -85,B 0,C 180,E1 -18826.64,E2 -18826.64} C_VEL
LIN {X 0,Y 253.215,Z 529.514,A -85,B 0,C 180,E1 -18828.613,E2 -18828.613} C_VEL
LIN {X 0,Y 255.042,Z 522.241,A -85,B 0,C 180,E1 -18830.58,E2 -18830.58} C_VEL
LIN {X 0,Y 257.307,Z 513.499,A -85,B 0,C 180,E1 -18832.482,E2 -18832.482} C_VEL
LIN {X 0,Y 259.575,Z 503.881,A -85,B 0,C 180,E1 -18834.174,E2 -18834.174} C_VEL
LIN {X 0,Y 261.589,Z 494.861,A -85,B 0,C 180,E1 -18835.459,E2 -18835.459} C_VEL
LIN {X 0,Y 263.363,Z 485.526,A -85,B 0,C 180,E1 -18836.55,E2 -18836.55} C_VEL
LIN {X 0,Y 265.061,Z 474.785,A -85,B 0,C 180,E1 -18837.539,E2 -18837.539} C_VEL
LIN {X 0,Y 266.451,Z 463.94,A -85,B 0,C 180,E1 -18838.291,E2 -18838.291} C_VEL
LIN {X 0,Y 267.581,Z 452.583,A -85,B 0,C 180,E1 -18838.836,E2 -18838.836} C_VEL
LIN {X 0,Y 268.384,Z 434.261,A -85,B 0,C 180,E1 -18839.414,E2 -18839.414} C_VEL
LIN {X 0,Y 270.146,Z 390.561,A -85,B 0,C 180,E1 -18840.61,E2 -18840.61} C_VEL
LIN {X 0,Y 267.872,Z 375.827,A -85,B 0,C 180,E1 -18841.447,E2 -18841.447} C_VEL
LIN {X 0,Y 261.942,Z 361.904,A -85,B 0,C 180,E1 -18842.87,E2 -18842.87} C_VEL
LIN {X 0,Y 255.444,Z 349.079,A -85,B 0,C 180,E1 -18844.469,E2 -18844.469} C_VEL
LIN {X 0,Y 251.913,Z 342.355,A -85,B 0,C 180,E1 -18845.437,E2 -18845.437} C_VEL
LIN {X 0,Y 250.584,Z 337.512,A -85,B 0,C 180,E1 -18847.6,E2 -18847.6} C_VEL
LIN {X 0,Y 249.021,Z 332.018,A -85,B 0,C 180,E1 -18850.475,E2 -18850.475} C_VEL
LIN {X 0,Y 248.984,Z 331.97,A -85,B 0,C 180,E1 -18854.883,E2 -18854.883} C_VEL
LIN {X 0,Y 249.008,Z 331.968,A -85,B 0,C 180,E1 -18857.362,E2 -18857.362} C_VEL
LIN {X 0,Y 249.024,Z 331.959,A -85,B 0,C 180,E1 -18861.62,E2 -18861.62} C_VEL
LIN {X 0,Y 249.043,Z 331.956,A -85,B 0,C 180,E1 -18865.64,E2 -18865.64} C_VEL
LIN {X 0,Y 249.05,Z 331.956,A -85,B 0,C 180,E1 -18869.473,E2 -18869.473} C_VEL
LIN {X 0,Y 249.072,Z 331.95,A -85,B 0,C 180,E1 -18873.163,E2 -18873.163} C_VEL
LIN {X 0,Y 249.079,Z 331.947,A -85,B 0,C 180,E1 -18876.733,E2 -18876.733} C_VEL
LIN {X 0,Y 249.111,Z 331.951,A -85,B 0,C 180,E1 -18880.212,E2 -18880.212} C_VEL
LIN {X 0,Y 249.242,Z 331.939,A -85,B 0,C 180,E1 -18883.622,E2 -18883.622} C_VEL
LIN {X 0,Y 249.254,Z 331.936,A -85,B 0,C 180,E1 -18888.617,E2 -18888.617} C_VEL
LIN {X 0,Y 249.486,Z 331.896,A -85,B 0,C 180,E1 -18891.903,E2 -18891.903} C_VEL
LIN {X 0,Y 249.438,Z 331.904,A -85,B 0,C 180,E1 -18896.77,E2 -18896.77} C_VEL
LIN {X 0,Y 249.73,Z 331.866,A -85,B 0,C 180,E1 -18900,E2 -18900} C_VEL
LIN {X 0,Y 249.438,Z 331.912,A -85,B 0,C 180,E1 -18903.231,E2 -18903.231} C_VEL
LIN {X 0,Y 249.486,Z 331.902,A -85,B 0,C 180,E1 -18908.097,E2 -18908.097} C_VEL
LIN {X 0,Y 249.254,Z 331.935,A -85,B 0,C 180,E1 -18911.384,E2 -18911.384} C_VEL
LIN {X 0,Y 249.243,Z 331.932,A -85,B 0,C 180,E1 -18916.378,E2 -18916.378} C_VEL
LIN {X 0,Y 249.085,Z 331.954,A -85,B 0,C 180,E1 -18921.519,E2 -18921.519} C_VEL
LIN {X 0,Y 249.113,Z 331.956,A -85,B 0,C 180,E1 -18925.474,E2 -18925.474} C_VEL
LIN {X 0,Y 249.116,Z 332.13,A -85,B 0,C 180,E1 -18927.971,E2 -18927.971} C_VEL
LIN {X 0,Y 250.453,Z 336.877,A -85,B 0,C 180,E1 -18930.287,E2 -18930.287} C_VEL
LIN {X 0,Y 252.548,Z 340.707,A -85,B 0,C 180,E1 -18930.928,E2 -18930.928} C_VEL
LIN {X 0,Y 259.185,Z 352.492,A -85,B 0,C 180,E1 -18932.569,E2 -18932.569} C_VEL
LIN {X 0,Y 266.013,Z 366.675,A -85,B 0,C 180,E1 -18934.197,E2 -18934.197} C_VEL
LIN {X 0,Y 270.42,Z 378.044,A -85,B 0,C 180,E1 -18935.257,E2 -18935.257} C_VEL
LIN {X 0,Y 270.554,Z 382.1,A -85,B 0,C 180,E1 -18935.413,E2 -18935.413} C_VEL
LIN {X 0,Y 267.808,Z 443.352,A -85,B 0,C 180,E1 -18937.104,E2 -18937.104} C_VEL
LIN {X 0,Y 267.054,Z 453.294,A -85,B 0,C 180,E1 -18937.532,E2 -18937.532} C_VEL
LIN {X 0,Y 265.923,Z 463.647,A -85,B 0,C 180,E1 -18938.163,E2 -18938.163} C_VEL
LIN {X 0,Y 264.541,Z 473.905,A -85,B 0,C 180,E1 -18939.006,E2 -18939.006} C_VEL
LIN {X 0,Y 262.875,Z 483.691,A -85,B 0,C 180,E1 -18940.024,E2 -18940.024} C_VEL
LIN {X 0,Y 260.925,Z 493.697,A -85,B 0,C 180,E1 -18941.34,E2 -18941.34} C_VEL
LIN {X 0,Y 258.847,Z 503.014,A -85,B 0,C 180,E1 -18942.855,E2 -18942.855} C_VEL
LIN {X 0,Y 257.184,Z 509.839,A -85,B 0,C 180,E1 -18944.166,E2 -18944.166} C_VEL
LIN {X 0,Y 255.016,Z 517.83,A -85,B 0,C 180,E1 -18946.025,E2 -18946.025} C_VEL
LIN {X 0,Y 252.942,Z 525.291,A -85,B 0,C 180,E1 -18948.176,E2 -18948.176} C_VEL
LIN {X 0,Y 251.164,Z 531.66,A -85,B 0,C 180,E1 -18950.463,E2 -18950.463} C_VEL
LIN {X 0,Y 249.657,Z 536.809,A -85,B 0,C 180,E1 -18952.772,E2 -18952.772} C_VEL
LIN {X 0,Y 248.511,Z 540.882,A -85,B 0,C 180,E1 -18955.098,E2 -18955.098} C_VEL
LIN {X 0,Y 247.71,Z 543.936,A -85,B 0,C 180,E1 -18957.38,E2 -18957.38} C_VEL
LIN {X 0,Y 247.222,Z 545.75,A -85,B 0,C 180,E1 -18959.223,E2 -18959.223} C_VEL
LIN {X 0,Y 246.695,Z 547.515,A -85,B 0,C 180,E1 -18962.025,E2 -18962.025} C_VEL
LIN {X 0,Y 246.45,Z 548.073,A -85,B 0,C 180,E1 -18964.675,E2 -18964.675} C_VEL
LIN {X 0,Y 246.437,Z 547.766,A -85,B 0,C 180,E1 -18966.468,E2 -18966.468} C_VEL
LIN {X 0,Y 246.485,Z 547.088,A -85,B 0,C 180,E1 -18968.243,E2 -18968.243} C_VEL
LIN {X 0,Y 246.7,Z 545.962,A -85,B 0,C 180,E1 -18970.07,E2 -18970.07} C_VEL
LIN {X 0,Y 247.129,Z 543.386,A -85,B 0,C 180,E1 -18972.626,E2 -18972.626} C_VEL
LIN {X 0,Y 247.787,Z 539.65,A -85,B 0,C 180,E1 -18975.211,E2 -18975.211} C_VEL
LIN {X 0,Y 248.809,Z 533.702,A -85,B 0,C 180,E1 -18978.183,E2 -18978.183} C_VEL
LIN {X 0,Y 249.84,Z 528.393,A -85,B 0,C 180,E1 -18980.283,E2 -18980.283} C_VEL
LIN {X 0,Y 251.169,Z 521.951,A -85,B 0,C 180,E1 -18982.362,E2 -18982.362} C_VEL
LIN {X 0,Y 252.752,Z 514.147,A -85,B 0,C 180,E1 -18984.415,E2 -18984.415} C_VEL
LIN {X 0,Y 254.314,Z 505.926,A -85,B 0,C 180,E1 -18986.194,E2 -18986.194} C_VEL
LIN {X 0,Y 255.846,Z 497.885,A -85,B 0,C 180,E1 -18987.639,E2 -18987.639} C_VEL
LIN {X 0,Y 257.407,Z 488.557,A -85,B 0,C 180,E1 -18989.022,E2 -18989.022} C_VEL
LIN {X 0,Y 258.826,Z 479.044,A -85,B 0,C 180,E1 -18990.172,E2 -18990.172} C_VEL
LIN {X 0,Y 260.216,Z 468.083,A -85,B 0,C 180,E1 -18991.21,E2 -18991.21} C_VEL
LIN {X 0,Y 261.225,Z 456.773,A -85,B 0,C 180,E1 -18992.024,E2 -18992.024} C_VEL
LIN {X 0,Y 262.087,Z 446.324,A -85,B 0,C 180,E1 -18992.546,E2 -18992.546} C_VEL
LIN {X 0,Y 262.841,Z 428.846,A -85,B 0,C 180,E1 -18993.093,E2 -18993.093} C_VEL
LIN {X 0,Y 264.525,Z 376.979,A -85,B 0,C 180,E1 -18994.522,E2 -18994.522} C_VEL
LIN {X 0,Y 262.77,Z 367.438,A -85,B 0,C 180,E1 -18994.998,E2 -18994.998} C_VEL
LIN {X 0,Y 256.97,Z 352.635,A -85,B 0,C 180,E1 -18996.091,E2 -18996.091} C_VEL
LIN {X 0,Y 250.636,Z 337.322,A -85,B 0,C 180,E1 -18997.375,E2 -18997.375} C_VEL
LIN {X 0,Y 249.666,Z 333.167,A -85,B 0,C 180,E1 -18999.076,E2 -18999.076} C_VEL
LIN {X 0,Y 249.349,Z 331.956,A -85,B 0,C 180,E1 -18999.736,E2 -18999.736} C_VEL
LIN {X 0,Y 249.208,Z 331.938,A -85,B 0,C 180,E1 -19004.703,E2 -19004.703} C_VEL
LIN {X 0,Y 249.14,Z 331.945,A -85,B 0,C 180,E1 -19008.077,E2 -19008.077} C_VEL
LIN {X 0,Y 249.086,Z 331.958,A -85,B 0,C 180,E1 -19011.518,E2 -19011.518} C_VEL
LIN {X 0,Y 249.119,Z 331.954,A -85,B 0,C 180,E1 -19015.476,E2 -19015.476} C_VEL
LIN {X 0,Y 249.075,Z 331.945,A -85,B 0,C 180,E1 -19018.989,E2 -19018.989} C_VEL
LIN {X 0,Y 249.038,Z 331.96,A -85,B 0,C 180,E1 -19022.425,E2 -19022.425} C_VEL
LIN {X 0,Y 249.071,Z 331.955,A -85,B 0,C 180,E1 -19026.339,E2 -19026.339} C_VEL
LIN {X 0,Y 249.028,Z 331.947,A -85,B 0,C 180,E1 -19030.474,E2 -19030.474} C_VEL
LIN {X 0,Y 249.01,Z 331.967,A -85,B 0,C 180,E1 -19034.878,E2 -19034.878} C_VEL
LIN {X 0,Y 249.02,Z 331.959,A -85,B 0,C 180,E1 -19037.363,E2 -19037.363} C_VEL
LIN {X 0,Y 249.044,Z 331.943,A -85,B 0,C 180,E1 -19042.201,E2 -19042.201} C_VEL
LIN {X 0,Y 249.045,Z 331.962,A -85,B 0,C 180,E1 -19045.639,E2 -19045.639} C_VEL
LIN {X 0,Y 249.004,Z 331.932,A -85,B 0,C 180,E1 -19049.466,E2 -19049.466} C_VEL
LIN {X 0,Y 249.041,Z 331.948,A -85,B 0,C 180,E1 -19053.158,E2 -19053.158} C_VEL
LIN {X 0,Y 249.059,Z 331.959,A -85,B 0,C 180,E1 -19056.73,E2 -19056.73} C_VEL
LIN {X 0,Y 249.085,Z 331.923,A -85,B 0,C 180,E1 -19060.209,E2 -19060.209} C_VEL
LIN {X 0,Y 249.198,Z 331.91,A -85,B 0,C 180,E1 -19063.619,E2 -19063.619} C_VEL
LIN {X 0,Y 249.244,Z 331.935,A -85,B 0,C 180,E1 -19068.616,E2 -19068.616} C_VEL
LIN {X 0,Y 249.42,Z 331.883,A -85,B 0,C 180,E1 -19071.9,E2 -19071.9} C_VEL
LIN {X 0,Y 249.265,Z 331.901,A -85,B 0,C 180,E1 -19075.147,E2 -19075.147} C_VEL
LIN {X 0,Y 249.66,Z 331.883,A -85,B 0,C 180,E1 -19078.386,E2 -19078.386} C_VEL
LIN {X 0,Y 249.662,Z 331.876,A -85,B 0,C 180,E1 -19081.613,E2 -19081.613} C_VEL
LIN {X 0,Y 249.416,Z 331.893,A -85,B 0,C 180,E1 -19087.073,E2 -19087.073} C_VEL
LIN {X 0,Y 248.718,Z 331.997,A -85,B 0,C 180,E1 -19088.42,E2 -19088.42} C_VEL
LIN {X 0,Y 245.76,Z 332.371,A -85,B 0,C 180,E1 -19090.612,E2 -19090.612} C_VEL
LIN {X 0,Y 243.251,Z 332.675,A -85,B 0,C 180,E1 -19092.398,E2 -19092.398} C_VEL
LIN {X 0,Y 242.174,Z 332.791,A -85,B 0,C 180,E1 -19093.786,E2 -19093.786} C_VEL
LIN {X 0,Y 242.086,Z 332.797,A -85,B 0,C 180,E1 -19094.258,E2 -19094.258} C_VEL
LIN {X 0,Y 242.094,Z 332.809,A -85,B 0,C 180,E1 -19096.875,E2 -19096.875} C_VEL
LIN {X 0,Y 241.987,Z 332.826,A -85,B 0,C 180,E1 -19102.182,E2 -19102.182} C_VEL
LIN {X 0,Y 242.033,Z 332.826,A -85,B 0,C 180,E1 -19105.82,E2 -19105.82} C_VEL
LIN {X 0,Y 241.969,Z 332.835,A -85,B 0,C 180,E1 -19109.588,E2 -19109.588} C_VEL
LIN {X 0,Y 241.979,Z 332.84,A -85,B 0,C 180,E1 -19113.492,E2 -19113.492} C_VEL
LIN {X 0,Y 241.964,Z 332.83,A -85,B 0,C 180,E1 -19117.586,E2 -19117.586} C_VEL
LIN {X 0,Y 241.898,Z 332.843,A -85,B 0,C 180,E1 -19121.93,E2 -19121.93} C_VEL
LIN {X 0,Y 241.907,Z 332.846,A -85,B 0,C 180,E1 -19126.577,E2 -19126.577} C_VEL
LIN {X 0,Y 241.991,Z 332.839,A -85,B 0,C 180,E1 -19131.641,E2 -19131.641} C_VEL
LIN {X 0,Y 242.04,Z 332.962,A -85,B 0,C 180,E1 -19133.46,E2 -19133.46} C_VEL
LIN {X 0,Y 243.733,Z 340.436,A -85,B 0,C 180,E1 -19136.779,E2 -19136.779} C_VEL
LIN {X 0,Y 244.372,Z 343.414,A -85,B 0,C 180,E1 -19137.89,E2 -19137.89} C_VEL
LIN {X 0,Y 251.53,Z 361.005,A -85,B 0,C 180,E1 -19139.381,E2 -19139.381} C_VEL
LIN {X 0,Y 254.76,Z 369.698,A -85,B 0,C 180,E1 -19140.035,E2 -19140.035} C_VEL
LIN {X 0,Y 257.752,Z 390.211,A -85,B 0,C 180,E1 -19141.017,E2 -19141.017} C_VEL
LIN {X 0,Y 255.623,Z 450.039,A -85,B 0,C 180,E1 -19142.746,E2 -19142.746} C_VEL
LIN {X 0,Y 254.988,Z 459.531,A -85,B 0,C 180,E1 -19143.171,E2 -19143.171} C_VEL
LIN {X 0,Y 253.983,Z 469.955,A -85,B 0,C 180,E1 -19143.831,E2 -19143.831} C_VEL
LIN {X 0,Y 252.683,Z 480.079,A -85,B 0,C 180,E1 -19144.682,E2 -19144.682} C_VEL
LIN {X 0,Y 251.139,Z 490.642,A -85,B 0,C 180,E1 -19145.841,E2 -19145.841} C_VEL
LIN {X 0,Y 249.406,Z 500.554,A -85,B 0,C 180,E1 -19147.203,E2 -19147.203} C_VEL
LIN {X 0,Y 247.871,Z 508.826,A -85,B 0,C 180,E1 -19148.589,E2 -19148.589} C_VEL
LIN {X 0,Y 246.229,Z 517.536,A -85,B 0,C 180,E1 -19150.372,E2 -19150.372} C_VEL
LIN {X 0,Y 244.898,Z 524.348,A -85,B 0,C 180,E1 -19152.031,E2 -19152.031} C_VEL
LIN {X 0,Y 243.407,Z 531.336,A -85,B 0,C 180,E1 -19154.08,E2 -19154.08} C_VEL
LIN {X 0,Y 241.9,Z 538.14,A -85,B 0,C 180,E1 -19156.56,E2 -19156.56} C_VEL
LIN {X 0,Y 241.228,Z 541.998,A -85,B 0,C 180,E1 -19158.232,E2 -19158.232} C_VEL
LIN {X 0,Y 240.459,Z 546.64,A -85,B 0,C 180,E1 -19160.749,E2 -19160.749} C_VEL
LIN {X 0,Y 239.966,Z 550.156,A -85,B 0,C 180,E1 -19163.272,E2 -19163.272} C_VEL
LIN {X 0,Y 239.728,Z 553.209,A -85,B 0,C 180,E1 -19166.638,E2 -19166.638} C_VEL
LIN {X 0,Y 239.767,Z 554.174,A -85,B 0,C 180,E1 -19168.32,E2 -19168.32} C_VEL
LIN {X 0,Y 239.768,Z 554.811,A -85,B 0,C 180,E1 -19171.68,E2 -19171.68} C_VEL
LIN {X 0,Y 239.838,Z 553.769,A -85,B 0,C 180,E1 -19175.043,E2 -19175.043} C_VEL
LIN {X 0,Y 240.028,Z 552.771,A -85,B 0,C 180,E1 -19176.726,E2 -19176.726} C_VEL
LIN {X 0,Y 240.791,Z 549.267,A -85,B 0,C 180,E1 -19180.086,E2 -19180.086} C_VEL
LIN {X 0,Y 241.771,Z 545.529,A -85,B 0,C 180,E1 -19182.592,E2 -19182.592} C_VEL
LIN {X 0,Y 243.108,Z 540.675,A -85,B 0,C 180,E1 -19185.081,E2 -19185.081} C_VEL
LIN {X 0,Y 244.764,Z 535.722,A -85,B 0,C 180,E1 -19187.116,E2 -19187.116} C_VEL
LIN {X 0,Y 246.803,Z 528.357,A -85,B 0,C 180,E1 -19189.548,E2 -19189.548} C_VEL
LIN {X 0,Y 248.825,Z 520.912,A -85,B 0,C 180,E1 -19191.542,E2 -19191.542} C_VEL
LIN {X 0,Y 250.976,Z 512.894,A -85,B 0,C 180,E1 -19193.299,E2 -19193.299} C_VEL
LIN {X 0,Y 253.149,Z 504.39,A -85,B 0,C 180,E1 -19194.828,E2 -19194.828} C_VEL
LIN {X 0,Y 255.241,Z 495.501,A -85,B 0,C 180,E1 -19196.139,E2 -19196.139} C_VEL
LIN {X 0,Y 257.388,Z 484.516,A -85,B 0,C 180,E1 -19197.437,E2 -19197.437} C_VEL
LIN {X 0,Y 259.009,Z 474.728,A -85,B 0,C 180,E1 -19198.349,E2 -19198.349} C_VEL
LIN {X 0,Y 260.5,Z 463.263,A -85,B 0,C 180,E1 -19199.154,E2 -19199.154} C_VEL
LIN {X 0,Y 261.64,Z 452.483,A -85,B 0,C 180,E1 -19199.674,E2 -19199.674} C_VEL
LIN {X 0,Y 262.493,Z 433.73,A -85,B 0,C 180,E1 -19200.279,E2 -19200.279} C_VEL
LIN {X 0,Y 264.23,Z 391.03,A -85,B 0,C 180,E1 -19201.484,E2 -19201.484} C_VEL
LIN {X 0,Y 262.282,Z 378.512,A -85,B 0,C 180,E1 -19202.228,E2 -19202.228} C_VEL
LIN {X 0,Y 256.829,Z 365.57,A -85,B 0,C 180,E1 -19203.602,E2 -19203.602} C_VEL
LIN {X 0,Y 249.689,Z 351.252,A -85,B 0,C 180,E1 -19205.458,E2 -19205.458} C_VEL
LIN {X 0,Y 244.741,Z 342.409,A -85,B 0,C 180,E1 -19206.86,E2 -19206.86} C_VEL
LIN {X 0,Y 244.148,Z 340.569,A -85,B 0,C 180,E1 -19207.583,E2 -19207.583} C_VEL
LIN {X 0,Y 241.992,Z 332.908,A -85,B 0,C 180,E1 -19211.708,E2 -19211.708} C_VEL
LIN {X 0,Y 241.924,Z 332.848,A -85,B 0,C 180,E1 -19216.574,E2 -19216.574} C_VEL
LIN {X 0,Y 241.955,Z 332.846,A -85,B 0,C 180,E1 -19220.281,E2 -19220.281} C_VEL
LIN {X 0,Y 241.986,Z 332.834,A -85,B 0,C 180,E1 -19224.49,E2 -19224.49} C_VEL
LIN {X 0,Y 241.973,Z 332.834,A -85,B 0,C 180,E1 -19228.48,E2 -19228.48} C_VEL
LIN {X 0,Y 242.006,Z 332.829,A -85,B 0,C 180,E1 -19232.313,E2 -19232.313} C_VEL
LIN {X 0,Y 242.057,Z 332.826,A -85,B 0,C 180,E1 -19236.016,E2 -19236.016} C_VEL
LIN {X 0,Y 242.038,Z 332.835,A -85,B 0,C 180,E1 -19239.609,E2 -19239.609} C_VEL
LIN {X 0,Y 242.163,Z 332.817,A -85,B 0,C 180,E1 -19243.279,E2 -19243.279} C_VEL
LIN {X 0,Y 242.187,Z 332.818,A -85,B 0,C 180,E1 -19248.28,E2 -19248.28} C_VEL
LIN {X 0,Y 242.436,Z 332.772,A -85,B 0,C 180,E1 -19251.666,E2 -19251.666} C_VEL
LIN {X 0,Y 242.262,Z 332.798,A -85,B 0,C 180,E1 -19255.008,E2 -19255.008} C_VEL
LIN {X 0,Y 242.638,Z 332.762,A -85,B 0,C 180,E1 -19258.341,E2 -19258.341} C_VEL
LIN {X 0,Y 242.638,Z 332.755,A -85,B 0,C 180,E1 -19261.66,E2 -19261.66} C_VEL
LIN {X 0,Y 242.433,Z 332.786,A -85,B 0,C 180,E1 -19266.709,E2 -19266.709} C_VEL
LIN {X 0,Y 242.347,Z 332.793,A -85,B 0,C 180,E1 -19270.021,E2 -19270.021} C_VEL
LIN {X 0,Y 242.168,Z 332.817,A -85,B 0,C 180,E1 -19275.141,E2 -19275.141} C_VEL
LIN {X 0,Y 242.073,Z 332.827,A -85,B 0,C 180,E1 -19278.625,E2 -19278.625} C_VEL
LIN {X 0,Y 242.007,Z 332.835,A -85,B 0,C 180,E1 -19282.181,E2 -19282.181} C_VEL
LIN {X 0,Y 242.043,Z 332.924,A -85,B 0,C 180,E1 -19286.631,E2 -19286.631} C_VEL
LIN {X 0,Y 243.228,Z 336.977,A -85,B 0,C 180,E1 -19288.769,E2 -19288.769} C_VEL
LIN {X 0,Y 245.54,Z 341.12,A -85,B 0,C 180,E1 -19289.542,E2 -19289.542} C_VEL
LIN {X 0,Y 251.335,Z 351.005,A -85,B 0,C 180,E1 -19291.094,E2 -19291.094} C_VEL
LIN {X 0,Y 257.248,Z 362.538,A -85,B 0,C 180,E1 -19292.606,E2 -19292.606} C_VEL
LIN {X 0,Y 262.756,Z 375.008,A -85,B 0,C 180,E1 -19293.971,E2 -19293.971} C_VEL
LIN {X 0,Y 264.828,Z 380.809,A -85,B 0,C 180,E1 -19294.5,E2 -19294.5} C_VEL
LIN {X 0,Y 261.951,Z 442.61,A -85,B 0,C 180,E1 -19296.234,E2 -19296.234} C_VEL
LIN {X 0,Y 261.102,Z 453.042,A -85,B 0,C 180,E1 -19296.675,E2 -19296.675} C_VEL
LIN {X 0,Y 260.034,Z 462.991,A -85,B 0,C 180,E1 -19297.287,E2 -19297.287} C_VEL
LIN {X 0,Y 258.508,Z 473.592,A -85,B 0,C 180,E1 -19298.157,E2 -19298.157} C_VEL
LIN {X 0,Y 256.807,Z 483.387,A -85,B 0,C 180,E1 -19299.189,E2 -19299.189} C_VEL
LIN {X 0,Y 254.949,Z 492.636,A -85,B 0,C 180,E1 -19300.402,E2 -19300.402} C_VEL
LIN {X 0,Y 252.731,Z 502.34,A -85,B 0,C 180,E1 -19301.984,E2 -19301.984} C_VEL
LIN {X 0,Y 250.448,Z 511.018,A -85,B 0,C 180,E1 -19303.714,E2 -19303.714} C_VEL
LIN {X 0,Y 248.296,Z 518.514,A -85,B 0,C 180,E1 -19305.529,E2 -19305.529} C_VEL
LIN {X 0,Y 246.351,Z 525.257,A -85,B 0,C 180,E1 -19307.522,E2 -19307.522} C_VEL
LIN {X 0,Y 244.543,Z 531.302,A -85,B 0,C 180,E1 -19309.712,E2 -19309.712} C_VEL
LIN {X 0,Y 243.061,Z 536.165,A -85,B 0,C 180,E1 -19311.873,E2 -19311.873} C_VEL
LIN {X 0,Y 241.692,Z 540.754,A -85,B 0,C 180,E1 -19314.508,E2 -19314.508} C_VEL
LIN {X 0,Y 240.953,Z 543.271,A -85,B 0,C 180,E1 -19316.346,E2 -19316.346} C_VEL
LIN {X 0,Y 240.357,Z 545.203,A -85,B 0,C 180,E1 -19318.243,E2 -19318.243} C_VEL
LIN {X 0,Y 239.642,Z 547.514,A -85,B 0,C 180,E1 -19321.62,E2 -19321.62} C_VEL
LIN {X 0,Y 239.402,Z 548.057,A -85,B 0,C 180,E1 -19323.874,E2 -19323.874} C_VEL
LIN {X 0,Y 239.347,Z 547.997,A -85,B 0,C 180,E1 -19325.727,E2 -19325.727} C_VEL
LIN {X 0,Y 239.342,Z 547.565,A -85,B 0,C 180,E1 -19327.559,E2 -19327.559} C_VEL
LIN {X 0,Y 239.563,Z 546.237,A -85,B 0,C 180,E1 -19329.848,E2 -19329.848} C_VEL
LIN {X 0,Y 240.105,Z 543.152,A -85,B 0,C 180,E1 -19332.98,E2 -19332.98} C_VEL
LIN {X 0,Y 240.791,Z 539.296,A -85,B 0,C 180,E1 -19335.636,E2 -19335.636} C_VEL
LIN {X 0,Y 241.712,Z 534.231,A -85,B 0,C 180,E1 -19338.257,E2 -19338.257} C_VEL
LIN {X 0,Y 242.692,Z 529.38,A -85,B 0,C 180,E1 -19340.291,E2 -19340.291} C_VEL
LIN {X 0,Y 244.139,Z 522.678,A -85,B 0,C 180,E1 -19342.557,E2 -19342.557} C_VEL
LIN {X 0,Y 245.769,Z 514.993,A -85,B 0,C 180,E1 -19344.668,E2 -19344.668} C_VEL
LIN {X 0,Y 247.349,Z 506.987,A -85,B 0,C 180,E1 -19346.483,E2 -19346.483} C_VEL
LIN {X 0,Y 249.165,Z 497.78,A -85,B 0,C 180,E1 -19348.182,E2 -19348.182} C_VEL
LIN {X 0,Y 250.791,Z 488.404,A -85,B 0,C 180,E1 -19349.599,E2 -19349.599} C_VEL
LIN {X 0,Y 252.256,Z 478.891,A -85,B 0,C 180,E1 -19350.768,E2 -19350.768} C_VEL
LIN {X 0,Y 253.609,Z 468.43,A -85,B 0,C 180,E1 -19351.787,E2 -19351.787} C_VEL
LIN {X 0,Y 254.673,Z 457.186,A -85,B 0,C 180,E1 -19352.62,E2 -19352.62} C_VEL
LIN {X 0,Y 255.552,Z 446.93,A -85,B 0,C 180,E1 -19353.153,E2 -19353.153} C_VEL
LIN {X 0,Y 256.368,Z 428.65,A -85,B 0,C 180,E1 -19353.741,E2 -19353.741} C_VEL
LIN {X 0,Y 258.083,Z 377.736,A -85,B 0,C 180,E1 -19355.174,E2 -19355.174} C_VEL
LIN {X 0,Y 256.541,Z 369.602,A -85,B 0,C 180,E1 -19355.599,E2 -19355.599} C_VEL
LIN {X 0,Y 250.598,Z 354.492,A -85,B 0,C 180,E1 -19356.767,E2 -19356.767} C_VEL
LIN {X 0,Y 244.024,Z 339.03,A -85,B 0,C 180,E1 -19358.097,E2 -19358.097} C_VEL
LIN {X 0,Y 243.318,Z 337.029,A -85,B 0,C 180,E1 -19358.364,E2 -19358.364} C_VEL
LIN {X 0,Y 242.263,Z 332.837,A -85,B 0,C 180,E1 -19360.341,E2 -19360.341} C_VEL
LIN {X 0,Y 242.169,Z 332.813,A -85,B 0,C 180,E1 -19365.141,E2 -19365.141} C_VEL
LIN {X 0,Y 242.074,Z 332.822,A -85,B 0,C 180,E1 -19368.624,E2 -19368.624} C_VEL
LIN {X 0,Y 242.009,Z 332.832,A -85,B 0,C 180,E1 -19372.181,E2 -19372.181} C_VEL
LIN {X 0,Y 242.069,Z 332.832,A -85,B 0,C 180,E1 -19375.838,E2 -19375.838} C_VEL
LIN {X 0,Y 242.009,Z 332.83,A -85,B 0,C 180,E1 -19379.583,E2 -19379.583} C_VEL
LIN {X 0,Y 241.993,Z 332.823,A -85,B 0,C 180,E1 -19383.491,E2 -19383.491} C_VEL
LIN {X 0,Y 242.004,Z 332.841,A -85,B 0,C 180,E1 -19387.579,E2 -19387.579} C_VEL
LIN {X 0,Y 241.946,Z 332.821,A -85,B 0,C 180,E1 -19391.921,E2 -19391.921} C_VEL
LIN {X 0,Y 241.939,Z 332.847,A -85,B 0,C 180,E1 -19396.571,E2 -19396.571} C_VEL
LIN {X 0,Y 241.958,Z 332.812,A -85,B 0,C 180,E1 -19400.281,E2 -19400.281} C_VEL
LIN {X 0,Y 241.989,Z 332.838,A -85,B 0,C 180,E1 -19404.489,E2 -19404.489} C_VEL
LIN {X 0,Y 241.955,Z 332.824,A -85,B 0,C 180,E1 -19408.477,E2 -19408.477} C_VEL
LIN {X 0,Y 241.972,Z 332.813,A -85,B 0,C 180,E1 -19412.308,E2 -19412.308} C_VEL
LIN {X 0,Y 242.038,Z 332.835,A -85,B 0,C 180,E1 -19416.014,E2 -19416.014} C_VEL
LIN {X 0,Y 242.022,Z 332.813,A -85,B 0,C 180,E1 -19419.606,E2 -19419.606} C_VEL
LIN {X 0,Y 242.118,Z 332.786,A -85,B 0,C 180,E1 -19423.316,E2 -19423.316} C_VEL
LIN {X 0,Y 242.156,Z 332.815,A -85,B 0,C 180,E1 -19426.574,E2 -19426.574} C_VEL
LIN {X 0,Y 242.344,Z 332.784,A -85,B 0,C 180,E1 -19430.404,E2 -19430.404} C_VEL
LIN {X 0,Y 242.399,Z 332.745,A -85,B 0,C 180,E1 -19433.34,E2 -19433.34} C_VEL
LIN {X 0,Y 242.62,Z 332.759,A -85,B 0,C 180,E1 -19438.34,E2 -19438.34} C_VEL
LIN {X 0,Y 242.622,Z 332.753,A -85,B 0,C 180,E1 -19441.659,E2 -19441.659} C_VEL
LIN {X 0,Y 242.386,Z 332.768,A -85,B 0,C 180,E1 -19447.056,E2 -19447.056} C_VEL
LIN {X 0,Y 242.266,Z 332.806,A -85,B 0,C 180,E1 -19450.023,E2 -19450.023} C_VEL
LIN {X 0,Y 242.086,Z 332.797,A -85,B 0,C 180,E1 -19454.258,E2 -19454.258} C_VEL
LIN {X 0,Y 241.4,Z 332.884,A -85,B 0,C 180,E1 -19455.646,E2 -19455.646} C_VEL
LIN {X 0,Y 238.487,Z 333.268,A -85,B 0,C 180,E1 -19457.908,E2 -19457.908} C_VEL
LIN {X 0,Y 236.036,Z 333.584,A -85,B 0,C 180,E1 -19459.752,E2 -19459.752} C_VEL
LIN {X 0,Y 235.016,Z 333.706,A -85,B 0,C 180,E1 -19461.185,E2 -19461.185} C_VEL
LIN {X 0,Y 234.95,Z 333.707,A -85,B 0,C 180,E1 -19461.67,E2 -19461.67} C_VEL
LIN {X 0,Y 234.969,Z 333.708,A -85,B 0,C 180,E1 -19466.193,E2 -19466.193} C_VEL
LIN {X 0,Y 234.899,Z 333.707,A -85,B 0,C 180,E1 -19470.572,E2 -19470.572} C_VEL
LIN {X 0,Y 234.922,Z 333.722,A -85,B 0,C 180,E1 -19474.639,E2 -19474.639} C_VEL
LIN {X 0,Y 234.911,Z 333.719,A -85,B 0,C 180,E1 -19478.935,E2 -19478.935} C_VEL
LIN {X 0,Y 234.858,Z 333.728,A -85,B 0,C 180,E1 -19484.095,E2 -19484.095} C_VEL
LIN {X 0,Y 234.859,Z 333.729,A -85,B 0,C 180,E1 -19488.426,E2 -19488.426} C_VEL
LIN {X 0,Y 234.984,Z 333.773,A -85,B 0,C 180,E1 -19492.724,E2 -19492.724} C_VEL
LIN {X 0,Y 236.824,Z 342.044,A -85,B 0,C 180,E1 -19496.542,E2 -19496.542} C_VEL
LIN {X 0,Y 237.096,Z 343.185,A -85,B 0,C 180,E1 -19496.931,E2 -19496.931} C_VEL
LIN {X 0,Y 244.551,Z 361.11,A -85,B 0,C 180,E1 -19498.558,E2 -19498.558} C_VEL
LIN {X 0,Y 248.689,Z 372.453,A -85,B 0,C 180,E1 -19499.435,E2 -19499.435} C_VEL
LIN {X 0,Y 251.339,Z 391.241,A -85,B 0,C 180,E1 -19500.358,E2 -19500.358} C_VEL
LIN {X 0,Y 249.149,Z 449.86,A -85,B 0,C 180,E1 -19502.09,E2 -19502.09} C_VEL
LIN {X 0,Y 248.503,Z 459.381,A -85,B 0,C 180,E1 -19502.526,E2 -19502.526} C_VEL
LIN {X 0,Y 247.459,Z 469.817,A -85,B 0,C 180,E1 -19503.201,E2 -19503.201} C_VEL
LIN {X 0,Y 246.238,Z 479.01,A -85,B 0,C 180,E1 -19503.971,E2 -19503.971} C_VEL
LIN {X 0,Y 244.648,Z 489.768,A -85,B 0,C 180,E1 -19505.157,E2 -19505.157} C_VEL
LIN {X 0,Y 242.851,Z 499.821,A -85,B 0,C 180,E1 -19506.552,E2 -19506.552} C_VEL
LIN {X 0,Y 241.011,Z 509.232,A -85,B 0,C 180,E1 -19508.173,E2 -19508.173} C_VEL
LIN {X 0,Y 239.329,Z 517.833,A -85,B 0,C 180,E1 -19509.998,E2 -19509.998} C_VEL
LIN {X 0,Y 237.764,Z 525.323,A -85,B 0,C 180,E1 -19511.918,E2 -19511.918} C_VEL
LIN {X 0,Y 236.254,Z 532.128,A -85,B 0,C 180,E1 -19514.028,E2 -19514.028} C_VEL
LIN {X 0,Y 234.966,Z 537.803,A -85,B 0,C 180,E1 -19516.155,E2 -19516.155} C_VEL
LIN {X 0,Y 233.932,Z 543.302,A -85,B 0,C 180,E1 -19518.739,E2 -19518.739} C_VEL
LIN {X 0,Y 233.22,Z 547.602,A -85,B 0,C 180,E1 -19521.334,E2 -19521.334} C_VEL
LIN {X 0,Y 232.905,Z 549.926,A -85,B 0,C 180,E1 -19523.067,E2 -19523.067} C_VEL
LIN {X 0,Y 232.641,Z 553.051,A -85,B 0,C 180,E1 -19526.536,E2 -19526.536} C_VEL
LIN {X 0,Y 232.663,Z 554.016,A -85,B 0,C 180,E1 -19528.269,E2 -19528.269} C_VEL
LIN {X 0,Y 232.715,Z 554.502,A -85,B 0,C 180,E1 -19530,E2 -19530} C_VEL
LIN {X 0,Y 232.665,Z 554.729,A -85,B 0,C 180,E1 -19531.731,E2 -19531.731} C_VEL
LIN {X 0,Y 232.764,Z 553.731,A -85,B 0,C 180,E1 -19535.197,E2 -19535.197} C_VEL
LIN {X 0,Y 232.974,Z 552.746,A -85,B 0,C 180,E1 -19536.93,E2 -19536.93} C_VEL
LIN {X 0,Y 233.782,Z 549.315,A -85,B 0,C 180,E1 -19540.391,E2 -19540.391} C_VEL
LIN {X 0,Y 234.829,Z 545.622,A -85,B 0,C 180,E1 -19542.971,E2 -19542.971} C_VEL
LIN {X 0,Y 236.26,Z 540.817,A -85,B 0,C 180,E1 -19545.529,E2 -19545.529} C_VEL
LIN {X 0,Y 238.298,Z 534.745,A -85,B 0,C 180,E1 -19548.039,E2 -19548.039} C_VEL
LIN {X 0,Y 240.1,Z 528.614,A -85,B 0,C 180,E1 -19550.117,E2 -19550.117} C_VEL
LIN {X 0,Y 242.25,Z 521.255,A -85,B 0,C 180,E1 -19552.157,E2 -19552.157} C_VEL
LIN {X 0,Y 244.747,Z 512.327,A -85,B 0,C 180,E1 -19554.154,E2 -19554.154} C_VEL
LIN {X 0,Y 247.038,Z 503.747,A -85,B 0,C 180,E1 -19555.712,E2 -19555.712} C_VEL
LIN {X 0,Y 249.212,Z 494.761,A -85,B 0,C 180,E1 -19557.048,E2 -19557.048} C_VEL
LIN {X 0,Y 251.153,Z 485.471,A -85,B 0,C 180,E1 -19558.178,E2 -19558.178} C_VEL
LIN {X 0,Y 253.012,Z 474.797,A -85,B 0,C 180,E1 -19559.199,E2 -19559.199} C_VEL
LIN {X 0,Y 254.565,Z 463.416,A -85,B 0,C 180,E1 -19560.015,E2 -19560.015} C_VEL
LIN {X 0,Y 255.768,Z 452.241,A -85,B 0,C 180,E1 -19560.564,E2 -19560.564} C_VEL
LIN {X 0,Y 256.649,Z 434.238,A -85,B 0,C 180,E1 -19561.154,E2 -19561.154} C_VEL
LIN {X 0,Y 258.448,Z 392.199,A -85,B 0,C 180,E1 -19562.363,E2 -19562.363} C_VEL
LIN {X 0,Y 256.697,Z 381.024,A -85,B 0,C 180,E1 -19563.057,E2 -19563.057} C_VEL
LIN {X 0,Y 250.864,Z 367.204,A -85,B 0,C 180,E1 -19564.62,E2 -19564.62} C_VEL
LIN {X 0,Y 244.862,Z 355.337,A -85,B 0,C 180,E1 -19566.261,E2 -19566.261} C_VEL
LIN {X 0,Y 239.413,Z 345.796,A -85,B 0,C 180,E1 -19567.835,E2 -19567.835} C_VEL
LIN {X 0,Y 237.324,Z 341.881,A -85,B 0,C 180,E1 -19568.563,E2 -19568.563} C_VEL
LIN {X 0,Y 235.556,Z 335.849,A -85,B 0,C 180,E1 -19571.765,E2 -19571.765} C_VEL
LIN {X 0,Y 234.882,Z 333.751,A -85,B 0,C 180,E1 -19573.171,E2 -19573.171} C_VEL
LIN {X 0,Y 234.877,Z 333.725,A -85,B 0,C 180,E1 -19576.512,E2 -19576.512} C_VEL
LIN {X 0,Y 234.917,Z 333.717,A -85,B 0,C 180,E1 -19581.079,E2 -19581.079} C_VEL
LIN {X 0,Y 234.929,Z 333.713,A -85,B 0,C 180,E1 -19585.362,E2 -19585.362} C_VEL
LIN {X 0,Y 234.93,Z 333.714,A -85,B 0,C 180,E1 -19589.433,E2 -19589.433} C_VEL
LIN {X 0,Y 234.994,Z 333.708,A -85,B 0,C 180,E1 -19593.794,E2 -19593.794} C_VEL
LIN {X 0,Y 235.012,Z 333.711,A -85,B 0,C 180,E1 -19598.97,E2 -19598.97} C_VEL
LIN {X 0,Y 235.097,Z 333.695,A -85,B 0,C 180,E1 -19603.06,E2 -19603.06} C_VEL
LIN {X 0,Y 235.147,Z 333.689,A -85,B 0,C 180,E1 -19607.924,E2 -19607.924} C_VEL
LIN {X 0,Y 235.392,Z 333.649,A -85,B 0,C 180,E1 -19611.415,E2 -19611.415} C_VEL
LIN {X 0,Y 235.407,Z 333.661,A -85,B 0,C 180,E1 -19613.142,E2 -19613.142} C_VEL
LIN {X 0,Y 235.598,Z 333.639,A -85,B 0,C 180,E1 -19618.291,E2 -19618.291} C_VEL
LIN {X 0,Y 235.598,Z 333.632,A -85,B 0,C 180,E1 -19621.71,E2 -19621.71} C_VEL
LIN {X 0,Y 235.407,Z 333.663,A -85,B 0,C 180,E1 -19626.859,E2 -19626.859} C_VEL
LIN {X 0,Y 235.255,Z 333.68,A -85,B 0,C 180,E1 -19630.326,E2 -19630.326} C_VEL
LIN {X 0,Y 235.115,Z 333.692,A -85,B 0,C 180,E1 -19635.607,E2 -19635.607} C_VEL
LIN {X 0,Y 235.008,Z 333.705,A -85,B 0,C 180,E1 -19639.206,E2 -19639.206} C_VEL
LIN {X 0,Y 234.952,Z 333.717,A -85,B 0,C 180,E1 -19642.884,E2 -19642.884} C_VEL
LIN {X 0,Y 235.047,Z 333.925,A -85,B 0,C 180,E1 -19645.386,E2 -19645.386} C_VEL
LIN {X 0,Y 236.05,Z 337.269,A -85,B 0,C 180,E1 -19647.183,E2 -19647.183} C_VEL
LIN {X 0,Y 240.87,Z 345.359,A -85,B 0,C 180,E1 -19648.719,E2 -19648.719} C_VEL
LIN {X 0,Y 246.694,Z 355.307,A -85,B 0,C 180,E1 -19650.361,E2 -19650.361} C_VEL
LIN {X 0,Y 253.374,Z 368.664,A -85,B 0,C 180,E1 -19652.143,E2 -19652.143} C_VEL
LIN {X 0,Y 258.583,Z 381.171,A -85,B 0,C 180,E1 -19653.51,E2 -19653.51} C_VEL
LIN {X 0,Y 259.017,Z 382.292,A -85,B 0,C 180,E1 -19653.622,E2 -19653.622} C_VEL
LIN {X 0,Y 256.053,Z 443.284,A -85,B 0,C 180,E1 -19655.371,E2 -19655.371} C_VEL
LIN {X 0,Y 255.168,Z 453.629,A -85,B 0,C 180,E1 -19655.827,E2 -19655.827} C_VEL
LIN {X 0,Y 253.992,Z 463.76,A -85,B 0,C 180,E1 -19656.471,E2 -19656.471} C_VEL
LIN {X 0,Y 252.443,Z 474.021,A -85,B 0,C 180,E1 -19657.336,E2 -19657.336} C_VEL
LIN {X 0,Y 250.791,Z 483.165,A -85,B 0,C 180,E1 -19658.311,E2 -19658.311} C_VEL
LIN {X 0,Y 248.705,Z 493.073,A -85,B 0,C 180,E1 -19659.642,E2 -19659.642} C_VEL
LIN {X 0,Y 246.398,Z 502.603,A -85,B 0,C 180,E1 -19661.235,E2 -19661.235} C_VEL
LIN {X 0,Y 244.286,Z 510.41,A -85,B 0,C 180,E1 -19662.809,E2 -19662.809} C_VEL
LIN {X 0,Y 242.012,Z 517.959,A -85,B 0,C 180,E1 -19664.645,E2 -19664.645} C_VEL
LIN {X 0,Y 239.702,Z 525.462,A -85,B 0,C 180,E1 -19666.915,E2 -19666.915} C_VEL
LIN {X 0,Y 237.618,Z 532.039,A -85,B 0,C 180,E1 -19669.406,E2 -19669.406} C_VEL
LIN {X 0,Y 236.254,Z 536.262,A -85,B 0,C 180,E1 -19671.34,E2 -19671.34} C_VEL
LIN {X 0,Y 234.863,Z 540.648,A -85,B 0,C 180,E1 -19673.896,E2 -19673.896} C_VEL
LIN {X 0,Y 233.899,Z 543.729,A -85,B 0,C 180,E1 -19676.229,E2 -19676.229} C_VEL
LIN {X 0,Y 232.999,Z 546.396,A -85,B 0,C 180,E1 -19679.151,E2 -19679.151} C_VEL
LIN {X 0,Y 232.611,Z 547.513,A -85,B 0,C 180,E1 -19681.187,E2 -19681.187} C_VEL
LIN {X 0,Y 232.252,Z 548.227,A -85,B 0,C 180,E1 -19684.935,E2 -19684.935} C_VEL
LIN {X 0,Y 232.228,Z 547.862,A -85,B 0,C 180,E1 -19686.832,E2 -19686.832} C_VEL
LIN {X 0,Y 232.443,Z 546.48,A -85,B 0,C 180,E1 -19689.603,E2 -19689.603} C_VEL
LIN {X 0,Y 232.878,Z 543.984,A -85,B 0,C 180,E1 -19692.435,E2 -19692.435} C_VEL
LIN {X 0,Y 233.58,Z 540.253,A -85,B 0,C 180,E1 -19695.303,E2 -19695.303} C_VEL
LIN {X 0,Y 234.425,Z 535.702,A -85,B 0,C 180,E1 -19697.886,E2 -19697.886} C_VEL
LIN {X 0,Y 235.821,Z 529.068,A -85,B 0,C 180,E1 -19700.757,E2 -19700.757} C_VEL
LIN {X 0,Y 237.395,Z 521.897,A -85,B 0,C 180,E1 -19703.199,E2 -19703.199} C_VEL
LIN {X 0,Y 239.012,Z 514.603,A -85,B 0,C 180,E1 -19705.227,E2 -19705.227} C_VEL
LIN {X 0,Y 240.655,Z 506.584,A -85,B 0,C 180,E1 -19707.071,E2 -19707.071} C_VEL
LIN {X 0,Y 242.493,Z 497.619,A -85,B 0,C 180,E1 -19708.755,E2 -19708.755} C_VEL
LIN {X 0,Y 244.182,Z 488.183,A -85,B 0,C 180,E1 -19710.206,E2 -19710.206} C_VEL
LIN {X 0,Y 245.713,Z 478.322,A -85,B 0,C 180,E1 -19711.434,E2 -19711.434} C_VEL
LIN {X 0,Y 247.116,Z 467.798,A -85,B 0,C 180,E1 -19712.464,E2 -19712.464} C_VEL
LIN {X 0,Y 248.157,Z 457.399,A -85,B 0,C 180,E1 -19713.247,E2 -19713.247} C_VEL
LIN {X 0,Y 249.064,Z 446.939,A -85,B 0,C 180,E1 -19713.804,E2 -19713.804} C_VEL
LIN {X 0,Y 249.912,Z 428.739,A -85,B 0,C 180,E1 -19714.402,E2 -19714.402} C_VEL
LIN {X 0,Y 251.746,Z 379.537,A -85,B 0,C 180,E1 -19715.811,E2 -19715.811} C_VEL
LIN {X 0,Y 250.508,Z 372.274,A -85,B 0,C 180,E1 -19716.191,E2 -19716.191} C_VEL
LIN {X 0,Y 245.308,Z 358.886,A -85,B 0,C 180,E1 -19717.255,E2 -19717.255} C_VEL
LIN {X 0,Y 237.657,Z 340.79,A -85,B 0,C 180,E1 -19718.853,E2 -19718.853} C_VEL
LIN {X 0,Y 236.124,Z 337.386,A -85,B 0,C 180,E1 -19719.259,E2 -19719.259} C_VEL
LIN {X 0,Y 235.2,Z 333.826,A -85,B 0,C 180,E1 -19720.873,E2 -19720.873} C_VEL
LIN {X 0,Y 235.116,Z 333.691,A -85,B 0,C 180,E1 -19725.606,E2 -19725.606} C_VEL
LIN {X 0,Y 235.009,Z 333.701,A -85,B 0,C 180,E1 -19729.206,E2 -19729.206} C_VEL
LIN {X 0,Y 234.955,Z 333.706,A -85,B 0,C 180,E1 -19732.884,E2 -19732.884} C_VEL
LIN {X 0,Y 234.969,Z 333.711,A -85,B 0,C 180,E1 -19736.658,E2 -19736.658} C_VEL
LIN {X 0,Y 234.925,Z 333.72,A -85,B 0,C 180,E1 -19740.569,E2 -19740.569} C_VEL
LIN {X 0,Y 234.963,Z 333.695,A -85,B 0,C 180,E1 -19744.633,E2 -19744.633} C_VEL
LIN {X 0,Y 234.944,Z 333.717,A -85,B 0,C 180,E1 -19748.944,E2 -19748.944} C_VEL
LIN {X 0,Y 234.892,Z 333.712,A -85,B 0,C 180,E1 -19753.485,E2 -19753.485} C_VEL
LIN {X 0,Y 234.892,Z 333.725,A -85,B 0,C 180,E1 -19756.515,E2 -19756.515} C_VEL
LIN {X 0,Y 234.919,Z 333.689,A -85,B 0,C 180,E1 -19761.078,E2 -19761.078} C_VEL
LIN {X 0,Y 234.932,Z 333.722,A -85,B 0,C 180,E1 -19765.362,E2 -19765.362} C_VEL
LIN {X 0,Y 234.901,Z 333.687,A -85,B 0,C 180,E1 -19769.427,E2 -19769.427} C_VEL
LIN {X 0,Y 234.971,Z 333.703,A -85,B 0,C 180,E1 -19773.806,E2 -19773.806} C_VEL
LIN {X 0,Y 234.991,Z 333.696,A -85,B 0,C 180,E1 -19778.968,E2 -19778.968} C_VEL
LIN {X 0,Y 235.058,Z 333.662,A -85,B 0,C 180,E1 -19783.092,E2 -19783.092} C_VEL
LIN {X 0,Y 235.112,Z 333.696,A -85,B 0,C 180,E1 -19787.921,E2 -19787.921} C_VEL
LIN {X 0,Y 235.313,Z 333.644,A -85,B 0,C 180,E1 -19791.411,E2 -19791.411} C_VEL
LIN {X 0,Y 235.35,Z 333.623,A -85,B 0,C 180,E1 -19793.139,E2 -19793.139} C_VEL
LIN {X 0,Y 235.579,Z 333.635,A -85,B 0,C 180,E1 -19798.29,E2 -19798.29} C_VEL
LIN {X 0,Y 235.581,Z 333.628,A -85,B 0,C 180,E1 -19801.709,E2 -19801.709} C_VEL
LIN {X 0,Y 235.361,Z 333.642,A -85,B 0,C 180,E1 -19806.859,E2 -19806.859} C_VEL
LIN {X 0,Y 235.212,Z 333.685,A -85,B 0,C 180,E1 -19810.327,E2 -19810.327} C_VEL
LIN {X 0,Y 235.043,Z 333.673,A -85,B 0,C 180,E1 -19815.611,E2 -19815.611} C_VEL
LIN {X 0,Y 234.961,Z 333.716,A -85,B 0,C 180,E1 -19819.209,E2 -19819.209} C_VEL
LIN {X 0,Y 234.95,Z 333.707,A -85,B 0,C 180,E1 -19821.67,E2 -19821.67} C_VEL
LIN {X 0,Y 234.657,Z 333.737,A -85,B 0,C 180,E1 -19822.628,E2 -19822.628} C_VEL
LIN {X 0,Y 233.302,Z 333.904,A -85,B 0,C 180,E1 -19824.042,E2 -19824.042} C_VEL
LIN {X 0,Y 228.925,Z 334.469,A -85,B 0,C 180,E1 -19827.341,E2 -19827.341} C_VEL
LIN {X 0,Y 227.914,Z 334.591,A -85,B 0,C 180,E1 -19828.821,E2 -19828.821} C_VEL
LIN {X 0,Y 227.859,Z 334.592,A -85,B 0,C 180,E1 -19829.323,E2 -19829.323} C_VEL
LIN {X 0,Y 227.876,Z 334.599,A -85,B 0,C 180,E1 -19833.72,E2 -19833.72} C_VEL
LIN {X 0,Y 227.836,Z 334.591,A -85,B 0,C 180,E1 -19838.092,E2 -19838.092} C_VEL
LIN {X 0,Y 227.778,Z 334.6,A -85,B 0,C 180,E1 -19842.749,E2 -19842.749} C_VEL
LIN {X 0,Y 227.79,Z 334.608,A -85,B 0,C 180,E1 -19847.252,E2 -19847.252} C_VEL
LIN {X 0,Y 227.94,Z 334.754,A -85,B 0,C 180,E1 -19852.106,E2 -19852.106} C_VEL
LIN {X 0,Y 229.786,Z 342.78,A -85,B 0,C 180,E1 -19855.854,E2 -19855.854} C_VEL
LIN {X 0,Y 231.405,Z 346.603,A -85,B 0,C 180,E1 -19856.327,E2 -19856.327} C_VEL
LIN {X 0,Y 239.408,Z 365.986,A -85,B 0,C 180,E1 -19858.089,E2 -19858.089} C_VEL
LIN {X 0,Y 242.559,Z 374.78,A -85,B 0,C 180,E1 -19858.784,E2 -19858.784} C_VEL
LIN {X 0,Y 244.961,Z 392.069,A -85,B 0,C 180,E1 -19859.663,E2 -19859.663} C_VEL
LIN {X 0,Y 242.69,Z 449.572,A -85,B 0,C 180,E1 -19861.398,E2 -19861.398} C_VEL
LIN {X 0,Y 242.043,Z 459.162,A -85,B 0,C 180,E1 -19861.846,E2 -19861.846} C_VEL
LIN {X 0,Y 240.964,Z 469.629,A -85,B 0,C 180,E1 -19862.536,E2 -19862.536} C_VEL
LIN {X 0,Y 239.563,Z 479.778,A -85,B 0,C 180,E1 -19863.424,E2 -19863.424} C_VEL
LIN {X 0,Y 237.907,Z 490.364,A -85,B 0,C 180,E1 -19864.637,E2 -19864.637} C_VEL
LIN {X 0,Y 236.076,Z 500.296,A -85,B 0,C 180,E1 -19866.07,E2 -19866.07} C_VEL
LIN {X 0,Y 234.373,Z 508.577,A -85,B 0,C 180,E1 -19867.522,E2 -19867.522} C_VEL
LIN {X 0,Y 232.841,Z 516.453,A -85,B 0,C 180,E1 -19869.195,E2 -19869.195} C_VEL
LIN {X 0,Y 231.012,Z 524.842,A -85,B 0,C 180,E1 -19871.371,E2 -19871.371} C_VEL
LIN {X 0,Y 229.419,Z 531.714,A -85,B 0,C 180,E1 -19873.539,E2 -19873.539} C_VEL
LIN {X 0,Y 228.037,Z 537.446,A -85,B 0,C 180,E1 -19875.726,E2 -19875.726} C_VEL
LIN {X 0,Y 226.937,Z 542.999,A -85,B 0,C 180,E1 -19878.387,E2 -19878.387} C_VEL
LIN {X 0,Y 226.177,Z 547.349,A -85,B 0,C 180,E1 -19881.062,E2 -19881.062} C_VEL
LIN {X 0,Y 225.837,Z 549.676,A -85,B 0,C 180,E1 -19882.849,E2 -19882.849} C_VEL
LIN {X 0,Y 225.541,Z 552.887,A -85,B 0,C 180,E1 -19886.427,E2 -19886.427} C_VEL
LIN {X 0,Y 225.563,Z 553.853,A -85,B 0,C 180,E1 -19888.214,E2 -19888.214} C_VEL
LIN {X 0,Y 225.631,Z 554.381,A -85,B 0,C 180,E1 -19890,E2 -19890} C_VEL
LIN {X 0,Y 225.565,Z 554.641,A -85,B 0,C 180,E1 -19891.785,E2 -19891.785} C_VEL
LIN {X 0,Y 225.689,Z 553.693,A -85,B 0,C 180,E1 -19895.36,E2 -19895.36} C_VEL
LIN {X 0,Y 225.915,Z 552.712,A -85,B 0,C 180,E1 -19897.148,E2 -19897.148} C_VEL
LIN {X 0,Y 226.788,Z 549.362,A -85,B 0,C 180,E1 -19900.716,E2 -19900.716} C_VEL
LIN {X 0,Y 227.901,Z 545.718,A -85,B 0,C 180,E1 -19903.373,E2 -19903.373} C_VEL
LIN {X 0,Y 229.432,Z 540.973,A -85,B 0,C 180,E1 -19906.003,E2 -19906.003} C_VEL
LIN {X 0,Y 231.559,Z 534.971,A -85,B 0,C 180,E1 -19908.583,E2 -19908.583} C_VEL
LIN {X 0,Y 233.433,Z 528.923,A -85,B 0,C 180,E1 -19910.717,E2 -19910.717} C_VEL
LIN {X 0,Y 235.694,Z 521.643,A -85,B 0,C 180,E1 -19912.807,E2 -19912.807} C_VEL
LIN {X 0,Y 238.326,Z 512.808,A -85,B 0,C 180,E1 -19914.848,E2 -19914.848} C_VEL
LIN {X 0,Y 240.692,Z 504.346,A -85,B 0,C 180,E1 -19916.442,E2 -19916.442} C_VEL
LIN {X 0,Y 243.306,Z 494.021,A -85,B 0,C 180,E1 -19917.994,E2 -19917.994} C_VEL
LIN {X 0,Y 245.292,Z 484.581,A -85,B 0,C 180,E1 -19919.149,E2 -19919.149} C_VEL
LIN {X 0,Y 247.223,Z 473.684,A -85,B 0,C 180,E1 -19920.186,E2 -19920.186} C_VEL
LIN {X 0,Y 248.702,Z 463.466,A -85,B 0,C 180,E1 -19920.922,E2 -19920.922} C_VEL
LIN {X 0,Y 249.976,Z 451.861,A -85,B 0,C 180,E1 -19921.5,E2 -19921.5} C_VEL
LIN {X 0,Y 250.968,Z 432.338,A -85,B 0,C 180,E1 -19922.145,E2 -19922.145} C_VEL
LIN {X 0,Y 252.744,Z 393.356,A -85,B 0,C 180,E1 -19923.287,E2 -19923.287} C_VEL
LIN {X 0,Y 251.35,Z 383.91,A -85,B 0,C 180,E1 -19923.892,E2 -19923.892} C_VEL
LIN {X 0,Y 245.842,Z 370.817,A -85,B 0,C 180,E1 -19925.439,E2 -19925.439} C_VEL
LIN {X 0,Y 240.256,Z 359.569,A -85,B 0,C 180,E1 -19927.058,E2 -19927.058} C_VEL
LIN {X 0,Y 235.16,Z 350.556,A -85,B 0,C 180,E1 -19928.598,E2 -19928.598} C_VEL
LIN {X 0,Y 232.27,Z 345.799,A -85,B 0,C 180,E1 -19929.504,E2 -19929.504} C_VEL
LIN {X 0,Y 229.942,Z 341.764,A -85,B 0,C 180,E1 -19930.365,E2 -19930.365} C_VEL
LIN {X 0,Y 228.18,Z 336.074,A -85,B 0,C 180,E1 -19933.64,E2 -19933.64} C_VEL
LIN {X 0,Y 227.836,Z 334.626,A -85,B 0,C 180,E1 -19934.731,E2 -19934.731} C_VEL
LIN {X 0,Y 227.823,Z 334.605,A -85,B 0,C 180,E1 -19939.623,E2 -19939.623} C_VEL
LIN {X 0,Y 227.88,Z 334.593,A -85,B 0,C 180,E1 -19944.129,E2 -19944.129} C_VEL
LIN {X 0,Y 227.869,Z 334.591,A -85,B 0,C 180,E1 -19948.378,E2 -19948.378} C_VEL
LIN {X 0,Y 227.885,Z 334.587,A -85,B 0,C 180,E1 -19952.445,E2 -19952.445} C_VEL
LIN {X 0,Y 227.914,Z 334.584,A -85,B 0,C 180,E1 -19956.368,E2 -19956.368} C_VEL
LIN {X 0,Y 227.943,Z 334.586,A -85,B 0,C 180,E1 -19960.175,E2 -19960.175} C_VEL
LIN {X 0,Y 228.058,Z 334.577,A -85,B 0,C 180,E1 -19963.898,E2 -19963.898} C_VEL
LIN {X 0,Y 228.172,Z 334.56,A -85,B 0,C 180,E1 -19969.351,E2 -19969.351} C_VEL
LIN {X 0,Y 228.36,Z 334.539,A -85,B 0,C 180,E1 -19972.929,E2 -19972.929} C_VEL
LIN {X 0,Y 228.556,Z 334.516,A -85,B 0,C 180,E1 -19978.238,E2 -19978.238} C_VEL
LIN {X 0,Y 228.556,Z 334.509,A -85,B 0,C 180,E1 -19981.763,E2 -19981.763} C_VEL
LIN {X 0,Y 228.36,Z 334.541,A -85,B 0,C 180,E1 -19987.072,E2 -19987.072} C_VEL
LIN {X 0,Y 228.169,Z 334.564,A -85,B 0,C 180,E1 -19990.65,E2 -19990.65} C_VEL
LIN {X 0,Y 228.066,Z 334.577,A -85,B 0,C 180,E1 -19994.272,E2 -19994.272} C_VEL
LIN {X 0,Y 228.004,Z 334.584,A -85,B 0,C 180,E1 -19997.954,E2 -19997.954} C_VEL
LIN {X 0,Y 227.929,Z 334.591,A -85,B 0,C 180,E1 -20002.8,E2 -20002.8} C_VEL
LIN {X 0,Y 227.941,Z 334.842,A -85,B 0,C 180,E1 -20003.871,E2 -20003.871} C_VEL
LIN {X 0,Y 228.832,Z 337.461,A -85,B 0,C 180,E1 -20005.405,E2 -20005.405} C_VEL
LIN {X 0,Y 231.489,Z 341.79,A -85,B 0,C 180,E1 -20006.37,E2 -20006.37} C_VEL
LIN {X 0,Y 237.914,Z 352.199,A -85,B 0,C 180,E1 -20008.357,E2 -20008.357} C_VEL
LIN {X 0,Y 244.498,Z 364.258,A -85,B 0,C 180,E1 -20010.28,E2 -20010.28} C_VEL
LIN {X 0,Y 250.342,Z 376.918,A -85,B 0,C 180,E1 -20011.902,E2 -20011.902} C_VEL
LIN {X 0,Y 253.246,Z 384.212,A -85,B 0,C 180,E1 -20012.705,E2 -20012.705} C_VEL
LIN {X 0,Y 250.281,Z 443.33,A -85,B 0,C 180,E1 -20014.445,E2 -20014.445} C_VEL
LIN {X 0,Y 249.407,Z 453.106,A -85,B 0,C 180,E1 -20014.873,E2 -20014.873} C_VEL
LIN {X 0,Y 248.214,Z 463.168,A -85,B 0,C 180,E1 -20015.508,E2 -20015.508} C_VEL
LIN {X 0,Y 246.611,Z 473.529,A -85,B 0,C 180,E1 -20016.382,E2 -20016.382} C_VEL
LIN {X 0,Y 244.676,Z 483.676,A -85,B 0,C 180,E1 -20017.487,E2 -20017.487} C_VEL
LIN {X 0,Y 242.565,Z 493.247,A -85,B 0,C 180,E1 -20018.8,E2 -20018.8} C_VEL
LIN {X 0,Y 240.113,Z 502.885,A -85,B 0,C 180,E1 -20020.447,E2 -20020.447} C_VEL
LIN {X 0,Y 238.21,Z 509.77,A -85,B 0,C 180,E1 -20021.844,E2 -20021.844} C_VEL
LIN {X 0,Y 235.23,Z 519.053,A -85,B 0,C 180,E1 -20024.189,E2 -20024.189} C_VEL
LIN {X 0,Y 232.965,Z 526.025,A -85,B 0,C 180,E1 -20026.388,E2 -20026.388} C_VEL
LIN {X 0,Y 231.11,Z 531.623,A -85,B 0,C 180,E1 -20028.545,E2 -20028.545} C_VEL
LIN {X 0,Y 229.268,Z 536.877,A -85,B 0,C 180,E1 -20031.067,E2 -20031.067} C_VEL
LIN {X 0,Y 228.051,Z 540.548,A -85,B 0,C 180,E1 -20033.251,E2 -20033.251} C_VEL
LIN {X 0,Y 226.825,Z 544.124,A -85,B 0,C 180,E1 -20036.102,E2 -20036.102} C_VEL
LIN {X 0,Y 226.171,Z 545.936,A -85,B 0,C 180,E1 -20038.112,E2 -20038.112} C_VEL
LIN {X 0,Y 225.581,Z 547.515,A -85,B 0,C 180,E1 -20040.733,E2 -20040.733} C_VEL
LIN {X 0,Y 225.194,Z 548.36,A -85,B 0,C 180,E1 -20044.093,E2 -20044.093} C_VEL
LIN {X 0,Y 225.141,Z 548.09,A -85,B 0,C 180,E1 -20046.058,E2 -20046.058} C_VEL
LIN {X 0,Y 225.311,Z 546.714,A -85,B 0,C 180,E1 -20049.354,E2 -20049.354} C_VEL
LIN {X 0,Y 225.865,Z 543.805,A -85,B 0,C 180,E1 -20052.807,E2 -20052.807} C_VEL
LIN {X 0,Y 226.562,Z 540.123,A -85,B 0,C 180,E1 -20055.631,E2 -20055.631} C_VEL
LIN {X 0,Y 227.75,Z 534.226,A -85,B 0,C 180,E1 -20058.88,E2 -20058.88} C_VEL
LIN {X 0,Y 228.891,Z 528.967,A -85,B 0,C 180,E1 -20061.169,E2 -20061.169} C_VEL
LIN {X 0,Y 230.373,Z 522.578,A -85,B 0,C 180,E1 -20063.431,E2 -20063.431} C_VEL
LIN {X 0,Y 232.043,Z 515.397,A -85,B 0,C 180,E1 -20065.517,E2 -20065.517} C_VEL
LIN {X 0,Y 233.94,Z 506.45,A -85,B 0,C 180,E1 -20067.633,E2 -20067.633} C_VEL
LIN {X 0,Y 235.855,Z 497.434,A -85,B 0,C 180,E1 -20069.36,E2 -20069.36} C_VEL
LIN {X 0,Y 237.604,Z 487.941,A -85,B 0,C 180,E1 -20070.848,E2 -20070.848} C_VEL
LIN {X 0,Y 239.104,Z 478.654,A -85,B 0,C 180,E1 -20072.034,E2 -20072.034} C_VEL
LIN {X 0,Y 240.571,Z 468.094,A -85,B 0,C 180,E1 -20073.096,E2 -20073.096} C_VEL
LIN {X 0,Y 241.668,Z 457.587,A -85,B 0,C 180,E1 -20073.908,E2 -20073.908} C_VEL
LIN {X 0,Y 242.638,Z 446.235,A -85,B 0,C 180,E1 -20074.517,E2 -20074.517} C_VEL
LIN {X 0,Y 243.569,Z 426.964,A -85,B 0,C 180,E1 -20075.149,E2 -20075.149} C_VEL
LIN {X 0,Y 245.28,Z 379.457,A -85,B 0,C 180,E1 -20076.558,E2 -20076.558} C_VEL
LIN {X 0,Y 244.273,Z 374.462,A -85,B 0,C 180,E1 -20076.848,E2 -20076.848} C_VEL
LIN {X 0,Y 239.056,Z 360.944,A -85,B 0,C 180,E1 -20077.964,E2 -20077.964} C_VEL
LIN {X 0,Y 231.786,Z 343.844,A -85,B 0,C 180,E1 -20079.533,E2 -20079.533} C_VEL
LIN {X 0,Y 228.86,Z 337.564,A -85,B 0,C 180,E1 -20080.25,E2 -20080.25} C_VEL
LIN {X 0,Y 228.125,Z 334.679,A -85,B 0,C 180,E1 -20081.608,E2 -20081.608} C_VEL
LIN {X 0,Y 228.06,Z 334.571,A -85,B 0,C 180,E1 -20086.102,E2 -20086.102} C_VEL
LIN {X 0,Y 227.939,Z 334.584,A -85,B 0,C 180,E1 -20089.826,E2 -20089.826} C_VEL
LIN {X 0,Y 227.909,Z 334.584,A -85,B 0,C 180,E1 -20093.633,E2 -20093.633} C_VEL
LIN {X 0,Y 227.881,Z 334.585,A -85,B 0,C 180,E1 -20097.556,E2 -20097.556} C_VEL
LIN {X 0,Y 227.871,Z 334.599,A -85,B 0,C 180,E1 -20101.622,E2 -20101.622} C_VEL
LIN {X 0,Y 227.902,Z 334.583,A -85,B 0,C 180,E1 -20105.868,E2 -20105.868} C_VEL
LIN {X 0,Y 227.836,Z 334.586,A -85,B 0,C 180,E1 -20110.375,E2 -20110.375} C_VEL
LIN {X 0,Y 227.838,Z 334.604,A -85,B 0,C 180,E1 -20115.192,E2 -20115.192} C_VEL
LIN {X 0,Y 227.828,Z 334.573,A -85,B 0,C 180,E1 -20119.623,E2 -20119.623} C_VEL
LIN {X 0,Y 227.883,Z 334.595,A -85,B 0,C 180,E1 -20124.128,E2 -20124.128} C_VEL
LIN {X 0,Y 227.858,Z 334.579,A -85,B 0,C 180,E1 -20128.375,E2 -20128.375} C_VEL
LIN {X 0,Y 227.858,Z 334.571,A -85,B 0,C 180,E1 -20132.441,E2 -20132.441} C_VEL
LIN {X 0,Y 227.901,Z 334.597,A -85,B 0,C 180,E1 -20136.366,E2 -20136.366} C_VEL
LIN {X 0,Y 227.925,Z 334.556,A -85,B 0,C 180,E1 -20140.173,E2 -20140.173} C_VEL
LIN {X 0,Y 228.026,Z 334.548,A -85,B 0,C 180,E1 -20143.895,E2 -20143.895} C_VEL
LIN {X 0,Y 228.068,Z 334.576,A -85,B 0,C 180,E1 -20147.543,E2 -20147.543} C_VEL
LIN {X 0,Y 228.255,Z 334.526,A -85,B 0,C 180,E1 -20151.144,E2 -20151.144} C_VEL
LIN {X 0,Y 228.303,Z 334.501,A -85,B 0,C 180,E1 -20152.927,E2 -20152.927} C_VEL
LIN {X 0,Y 228.537,Z 334.512,A -85,B 0,C 180,E1 -20158.237,E2 -20158.237} C_VEL
LIN {X 0,Y 228.539,Z 334.503,A -85,B 0,C 180,E1 -20161.762,E2 -20161.762} C_VEL
LIN {X 0,Y 228.313,Z 334.521,A -85,B 0,C 180,E1 -20167.072,E2 -20167.072} C_VEL
LIN {X 0,Y 228.141,Z 334.566,A -85,B 0,C 180,E1 -20170.651,E2 -20170.651} C_VEL
LIN {X 0,Y 228.001,Z 334.553,A -85,B 0,C 180,E1 -20176.106,E2 -20176.106} C_VEL
LIN {X 0,Y 227.925,Z 334.582,A -85,B 0,C 180,E1 -20181.716,E2 -20181.716} C_VEL
LIN {X 0,Y 227.923,Z 334.588,A -85,B 0,C 180,E1 -20186.592,E2 -20186.592} C_VEL
LIN {X 0,Y 227.859,Z 334.592,A -85,B 0,C 180,E1 -20189.323,E2 -20189.323} C_VEL
LIN {X 0,Y 227.364,Z 334.656,A -85,B 0,C 180,E1 -20190.8,E2 -20190.8} C_VEL
LIN {X 0,Y 226.016,Z 334.825,A -85,B 0,C 180,E1 -20192.258,E2 -20192.258} C_VEL
LIN {X 0,Y 221.481,Z 335.388,A -85,B 0,C 180,E1 -20196.19,E2 -20196.19} C_VEL
LIN {X 0,Y 220.821,Z 335.463,A -85,B 0,C 180,E1 -20197.215,E2 -20197.215} C_VEL
LIN {X 0,Y 220.741,Z 335.477,A -85,B 0,C 180,E1 -20201.958,E2 -20201.958} C_VEL
LIN {X 0,Y 220.753,Z 335.483,A -85,B 0,C 180,E1 -20205.54,E2 -20205.54} C_VEL
LIN {X 0,Y 220.781,Z 335.485,A -85,B 0,C 180,E1 -20210.457,E2 -20210.457} C_VEL
LIN {X 0,Y 220.846,Z 335.622,A -85,B 0,C 180,E1 -20211.324,E2 -20211.324} C_VEL
LIN {X 0,Y 222.556,Z 342.745,A -85,B 0,C 180,E1 -20214.807,E2 -20214.807} C_VEL
LIN {X 0,Y 224.646,Z 347.725,A -85,B 0,C 180,E1 -20215.404,E2 -20215.404} C_VEL
LIN {X 0,Y 232.012,Z 365.008,A -85,B 0,C 180,E1 -20217.086,E2 -20217.086} C_VEL
LIN {X 0,Y 236.386,Z 376.612,A -85,B 0,C 180,E1 -20218.079,E2 -20218.079} C_VEL
LIN {X 0,Y 238.599,Z 393.112,A -85,B 0,C 180,E1 -20218.936,E2 -20218.936} C_VEL
LIN {X 0,Y 236.29,Z 449.287,A -85,B 0,C 180,E1 -20220.67,E2 -20220.67} C_VEL
LIN {X 0,Y 235.622,Z 458.942,A -85,B 0,C 180,E1 -20221.129,E2 -20221.129} C_VEL
LIN {X 0,Y 234.505,Z 469.44,A -85,B 0,C 180,E1 -20221.834,E2 -20221.834} C_VEL
LIN {X 0,Y 233.189,Z 478.669,A -85,B 0,C 180,E1 -20222.638,E2 -20222.638} C_VEL
LIN {X 0,Y 231.502,Z 489.457,A -85,B 0,C 180,E1 -20223.883,E2 -20223.883} C_VEL
LIN {X 0,Y 229.548,Z 499.528,A -85,B 0,C 180,E1 -20225.345,E2 -20225.345} C_VEL
LIN {X 0,Y 227.543,Z 508.954,A -85,B 0,C 180,E1 -20227.049,E2 -20227.049} C_VEL
LIN {X 0,Y 225.802,Z 517.365,A -85,B 0,C 180,E1 -20228.925,E2 -20228.925} C_VEL
LIN {X 0,Y 224.276,Z 524.36,A -85,B 0,C 180,E1 -20230.79,E2 -20230.79} C_VEL
LIN {X 0,Y 222.601,Z 531.299,A -85,B 0,C 180,E1 -20233.019,E2 -20233.019} C_VEL
LIN {X 0,Y 221.132,Z 537.09,A -85,B 0,C 180,E1 -20235.27,E2 -20235.27} C_VEL
LIN {X 0,Y 219.959,Z 542.697,A -85,B 0,C 180,E1 -20238.013,E2 -20238.013} C_VEL
LIN {X 0,Y 219.155,Z 547.096,A -85,B 0,C 180,E1 -20240.773,E2 -20240.773} C_VEL
LIN {X 0,Y 218.796,Z 549.424,A -85,B 0,C 180,E1 -20242.618,E2 -20242.618} C_VEL
LIN {X 0,Y 218.447,Z 552.724,A -85,B 0,C 180,E1 -20246.311,E2 -20246.311} C_VEL
LIN {X 0,Y 218.465,Z 553.69,A -85,B 0,C 180,E1 -20248.156,E2 -20248.156} C_VEL
LIN {X 0,Y 218.53,Z 554.26,A -85,B 0,C 180,E1 -20250,E2 -20250} C_VEL
LIN {X 0,Y 218.467,Z 554.544,A -85,B 0,C 180,E1 -20251.843,E2 -20251.843} C_VEL
LIN {X 0,Y 218.629,Z 553.657,A -85,B 0,C 180,E1 -20255.534,E2 -20255.534} C_VEL
LIN {X 0,Y 218.852,Z 552.677,A -85,B 0,C 180,E1 -20257.38,E2 -20257.38} C_VEL
LIN {X 0,Y 219.794,Z 549.427,A -85,B 0,C 180,E1 -20261.061,E2 -20261.061} C_VEL
LIN {X 0,Y 220.987,Z 545.839,A -85,B 0,C 180,E1 -20263.799,E2 -20263.799} C_VEL
LIN {X 0,Y 222.625,Z 541.15,A -85,B 0,C 180,E1 -20266.506,E2 -20266.506} C_VEL
LIN {X 0,Y 224.845,Z 535.21,A -85,B 0,C 180,E1 -20269.159,E2 -20269.159} C_VEL
LIN {X 0,Y 227.244,Z 527.817,A -85,B 0,C 180,E1 -20271.785,E2 -20271.785} C_VEL
LIN {X 0,Y 229.713,Z 520.334,A -85,B 0,C 180,E1 -20273.915,E2 -20273.915} C_VEL
LIN {X 0,Y 232.237,Z 512.273,A -85,B 0,C 180,E1 -20275.786,E2 -20275.786} C_VEL
LIN {X 0,Y 234.721,Z 503.741,A -85,B 0,C 180,E1 -20277.41,E2 -20277.41} C_VEL
LIN {X 0,Y 237.095,Z 494.817,A -85,B 0,C 180,E1 -20278.795,E2 -20278.795} C_VEL
LIN {X 0,Y 239.17,Z 485.618,A -85,B 0,C 180,E1 -20279.97,E2 -20279.97} C_VEL
LIN {X 0,Y 241.358,Z 473.891,A -85,B 0,C 180,E1 -20281.121,E2 -20281.121} C_VEL
LIN {X 0,Y 243.018,Z 462.929,A -85,B 0,C 180,E1 -20281.917,E2 -20281.917} C_VEL
LIN {X 0,Y 244.255,Z 452.121,A -85,B 0,C 180,E1 -20282.466,E2 -20282.466} C_VEL
LIN {X 0,Y 245.181,Z 434.961,A -85,B 0,C 180,E1 -20283.058,E2 -20283.058} C_VEL
LIN {X 0,Y 247.138,Z 394.421,A -85,B 0,C 180,E1 -20284.264,E2 -20284.264} C_VEL
LIN {X 0,Y 246.055,Z 386.849,A -85,B 0,C 180,E1 -20284.764,E2 -20284.764} C_VEL
LIN {X 0,Y 240.632,Z 373.875,A -85,B 0,C 180,E1 -20286.375,E2 -20286.375} C_VEL
LIN {X 0,Y 235.136,Z 362.809,A -85,B 0,C 180,E1 -20288.058,E2 -20288.058} C_VEL
LIN {X 0,Y 230.801,Z 355.033,A -85,B 0,C 180,E1 -20289.438,E2 -20289.438} C_VEL
LIN {X 0,Y 228.177,Z 350.659,A -85,B 0,C 180,E1 -20290.31,E2 -20290.31} C_VEL
LIN {X 0,Y 224.962,Z 345.613,A -85,B 0,C 180,E1 -20291.429,E2 -20291.429} C_VEL
LIN {X 0,Y 222.623,Z 341.52,A -85,B 0,C 180,E1 -20292.423,E2 -20292.423} C_VEL
LIN {X 0,Y 220.827,Z 335.885,A -85,B 0,C 180,E1 -20295.985,E2 -20295.985} C_VEL
LIN {X 0,Y 220.76,Z 335.485,A -85,B 0,C 180,E1 -20296.807,E2 -20296.807} C_VEL
LIN {X 0,Y 220.805,Z 335.478,A -85,B 0,C 180,E1 -20300.463,E2 -20300.463} C_VEL
LIN {X 0,Y 220.8,Z 335.472,A -85,B 0,C 180,E1 -20305.046,E2 -20305.046} C_VEL
LIN {X 0,Y 220.868,Z 335.465,A -85,B 0,C 180,E1 -20309.395,E2 -20309.395} C_VEL
LIN {X 0,Y 220.895,Z 335.461,A -85,B 0,C 180,E1 -20313.55,E2 -20313.55} C_VEL
LIN {X 0,Y 220.878,Z 335.46,A -85,B 0,C 180,E1 -20317.554,E2 -20317.554} C_VEL
LIN {X 0,Y 220.985,Z 335.448,A -85,B 0,C 180,E1 -20322.571,E2 -20322.571} C_VEL
LIN {X 0,Y 221.027,Z 335.44,A -85,B 0,C 180,E1 -20327.14,E2 -20327.14} C_VEL
LIN {X 0,Y 221.259,Z 335.409,A -85,B 0,C 180,E1 -20330.862,E2 -20330.862} C_VEL
LIN {X 0,Y 221.297,Z 335.414,A -85,B 0,C 180,E1 -20332.702,E2 -20332.702} C_VEL
LIN {X 0,Y 221.514,Z 335.393,A -85,B 0,C 180,E1 -20338.182,E2 -20338.182} C_VEL
LIN {X 0,Y 221.514,Z 335.387,A -85,B 0,C 180,E1 -20341.819,E2 -20341.819} C_VEL
LIN {X 0,Y 221.313,Z 335.416,A -85,B 0,C 180,E1 -20347.298,E2 -20347.298} C_VEL
LIN {X 0,Y 221.113,Z 335.444,A -85,B 0,C 180,E1 -20350.995,E2 -20350.995} C_VEL
LIN {X 0,Y 221.018,Z 335.448,A -85,B 0,C 180,E1 -20356.63,E2 -20356.63} C_VEL
LIN {X 0,Y 220.909,Z 335.508,A -85,B 0,C 180,E1 -20361.951,E2 -20361.951} C_VEL
LIN {X 0,Y 221.392,Z 337.397,A -85,B 0,C 180,E1 -20363.246,E2 -20363.246} C_VEL
LIN {X 0,Y 223.311,Z 340.703,A -85,B 0,C 180,E1 -20364.101,E2 -20364.101} C_VEL
LIN {X 0,Y 225.389,Z 343.497,A -85,B 0,C 180,E1 -20364.834,E2 -20364.834} C_VEL
LIN {X 0,Y 229.695,Z 350.351,A -85,B 0,C 180,E1 -20366.314,E2 -20366.314} C_VEL
LIN {X 0,Y 236.016,Z 361.105,A -85,B 0,C 180,E1 -20368.317,E2 -20368.317} C_VEL
LIN {X 0,Y 241.715,Z 372.407,A -85,B 0,C 180,E1 -20370.038,E2 -20370.038} C_VEL
LIN {X 0,Y 247.057,Z 384.734,A -85,B 0,C 180,E1 -20371.589,E2 -20371.589} C_VEL
LIN {X 0,Y 247.631,Z 387.05,A -85,B 0,C 180,E1 -20371.788,E2 -20371.788} C_VEL
LIN {X 0,Y 244.571,Z 443.612,A -85,B 0,C 180,E1 -20373.469,E2 -20373.469} C_VEL
LIN {X 0,Y 243.634,Z 453.646,A -85,B 0,C 180,E1 -20373.923,E2 -20373.923} C_VEL
LIN {X 0,Y 242.304,Z 464.135,A -85,B 0,C 180,E1 -20374.612,E2 -20374.612} C_VEL
LIN {X 0,Y 240.703,Z 473.925,A -85,B 0,C 180,E1 -20375.463,E2 -20375.463} C_VEL
LIN {X 0,Y 238.527,Z 484.767,A -85,B 0,C 180,E1 -20376.693,E2 -20376.693} C_VEL
LIN {X 0,Y 236.355,Z 493.995,A -85,B 0,C 180,E1 -20378.005,E2 -20378.005} C_VEL
LIN {X 0,Y 233.853,Z 503.274,A -85,B 0,C 180,E1 -20379.636,E2 -20379.636} C_VEL
LIN {X 0,Y 231.691,Z 510.638,A -85,B 0,C 180,E1 -20381.197,E2 -20381.197} C_VEL
LIN {X 0,Y 229.066,Z 518.544,A -85,B 0,C 180,E1 -20383.225,E2 -20383.225} C_VEL
LIN {X 0,Y 226.569,Z 525.746,A -85,B 0,C 180,E1 -20385.516,E2 -20385.516} C_VEL
LIN {X 0,Y 224.583,Z 531.393,A -85,B 0,C 180,E1 -20387.716,E2 -20387.716} C_VEL
LIN {X 0,Y 222.896,Z 535.964,A -85,B 0,C 180,E1 -20389.873,E2 -20389.873} C_VEL
LIN {X 0,Y 221.11,Z 540.831,A -85,B 0,C 180,E1 -20392.849,E2 -20392.849} C_VEL
LIN {X 0,Y 220.118,Z 543.431,A -85,B 0,C 180,E1 -20394.921,E2 -20394.921} C_VEL
LIN {X 0,Y 219.406,Z 545.411,A -85,B 0,C 180,E1 -20397.007,E2 -20397.007} C_VEL
LIN {X 0,Y 218.554,Z 547.526,A -85,B 0,C 180,E1 -20400.255,E2 -20400.255} C_VEL
LIN {X 0,Y 218.431,Z 547.964,A -85,B 0,C 180,E1 -20401.143,E2 -20401.143} C_VEL
LIN {X 0,Y 218.076,Z 548.456,A -85,B 0,C 180,E1 -20404.471,E2 -20404.471} C_VEL
LIN {X 0,Y 218.026,Z 547.912,A -85,B 0,C 180,E1 -20407.244,E2 -20407.244} C_VEL
LIN {X 0,Y 218.203,Z 546.862,A -85,B 0,C 180,E1 -20409.25,E2 -20409.25} C_VEL
LIN {X 0,Y 218.841,Z 543.574,A -85,B 0,C 180,E1 -20413.2,E2 -20413.2} C_VEL
LIN {X 0,Y 219.616,Z 539.753,A -85,B 0,C 180,E1 -20416.113,E2 -20416.113} C_VEL
LIN {X 0,Y 220.66,Z 534.722,A -85,B 0,C 180,E1 -20418.983,E2 -20418.983} C_VEL
LIN {X 0,Y 221.831,Z 529.55,A -85,B 0,C 180,E1 -20421.345,E2 -20421.345} C_VEL
LIN {X 0,Y 223.36,Z 523.257,A -85,B 0,C 180,E1 -20423.678,E2 -20423.678} C_VEL
LIN {X 0,Y 225.235,Z 515.438,A -85,B 0,C 180,E1 -20426.02,E2 -20426.02} C_VEL
LIN {X 0,Y 227.256,Z 506.312,A -85,B 0,C 180,E1 -20428.228,E2 -20428.228} C_VEL
LIN {X 0,Y 228.993,Z 498.527,A -85,B 0,C 180,E1 -20429.78,E2 -20429.78} C_VEL
LIN {X 0,Y 230.795,Z 489.245,A -85,B 0,C 180,E1 -20431.309,E2 -20431.309} C_VEL
LIN {X 0,Y 232.449,Z 479.565,A -85,B 0,C 180,E1 -20432.601,E2 -20432.601} C_VEL
LIN {X 0,Y 234.067,Z 468.35,A -85,B 0,C 180,E1 -20433.766,E2 -20433.766} C_VEL
LIN {X 0,Y 235.199,Z 457.795,A -85,B 0,C 180,E1 -20434.606,E2 -20434.606} C_VEL
LIN {X 0,Y 236.189,Z 446.857,A -85,B 0,C 180,E1 -20435.213,E2 -20435.213} C_VEL
LIN {X 0,Y 237.122,Z 428.707,A -85,B 0,C 180,E1 -20435.832,E2 -20435.832} C_VEL
LIN {X 0,Y 238.962,Z 380.612,A -85,B 0,C 180,E1 -20437.287,E2 -20437.287} C_VEL
LIN {X 0,Y 238.168,Z 376.893,A -85,B 0,C 180,E1 -20437.516,E2 -20437.516} C_VEL
LIN {X 0,Y 234.105,Z 366.225,A -85,B 0,C 180,E1 -20438.414,E2 -20438.414} C_VEL
LIN {X 0,Y 226.417,Z 347.748,A -85,B 0,C 180,E1 -20440.149,E2 -20440.149} C_VEL
LIN {X 0,Y 221.619,Z 337.8,A -85,B 0,C 180,E1 -20441.307,E2 -20441.307} C_VEL
LIN {X 0,Y 221.048,Z 335.595,A -85,B 0,C 180,E1 -20442.335,E2 -20442.335} C_VEL
LIN {X 0,Y 221.019,Z 335.452,A -85,B 0,C 180,E1 -20446.63,E2 -20446.63} C_VEL
LIN {X 0,Y 220.887,Z 335.468,A -85,B 0,C 180,E1 -20450.487,E2 -20450.487} C_VEL
LIN {X 0,Y 220.864,Z 335.466,A -85,B 0,C 180,E1 -20454.436,E2 -20454.436} C_VEL
LIN {X 0,Y 220.829,Z 335.461,A -85,B 0,C 180,E1 -20458.515,E2 -20458.515} C_VEL
LIN {X 0,Y 220.825,Z 335.467,A -85,B 0,C 180,E1 -20462.755,E2 -20462.755} C_VEL
LIN {X 0,Y 220.841,Z 335.475,A -85,B 0,C 180,E1 -20467.288,E2 -20467.288} C_VEL
LIN {X 0,Y 220.778,Z 335.456,A -85,B 0,C 180,E1 -20471.951,E2 -20471.951} C_VEL
LIN {X 0,Y 220.778,Z 335.483,A -85,B 0,C 180,E1 -20475.547,E2 -20475.547} C_VEL
LIN {X 0,Y 220.809,Z 335.444,A -85,B 0,C 180,E1 -20480.463,E2 -20480.463} C_VEL
LIN {X 0,Y 220.803,Z 335.479,A -85,B 0,C 180,E1 -20485.045,E2 -20485.045} C_VEL
LIN {X 0,Y 220.836,Z 335.438,A -85,B 0,C 180,E1 -20489.39,E2 -20489.39} C_VEL
LIN {X 0,Y 220.878,Z 335.457,A -85,B 0,C 180,E1 -20493.547,E2 -20493.547} C_VEL
LIN {X 0,Y 220.871,Z 335.468,A -85,B 0,C 180,E1 -20497.552,E2 -20497.552} C_VEL
LIN {X 0,Y 220.931,Z 335.416,A -85,B 0,C 180,E1 -20502.617,E2 -20502.617} C_VEL
LIN {X 0,Y 221.006,Z 335.453,A -85,B 0,C 180,E1 -20507.138,E2 -20507.138} C_VEL
LIN {X 0,Y 221.196,Z 335.408,A -85,B 0,C 180,E1 -20510.859,E2 -20510.859} C_VEL
LIN {X 0,Y 221.24,Z 335.381,A -85,B 0,C 180,E1 -20512.7,E2 -20512.7} C_VEL
LIN {X 0,Y 221.471,Z 335.391,A -85,B 0,C 180,E1 -20518.181,E2 -20518.181} C_VEL
LIN {X 0,Y 221.472,Z 335.382,A -85,B 0,C 180,E1 -20521.818,E2 -20521.818} C_VEL
LIN {X 0,Y 221.25,Z 335.403,A -85,B 0,C 180,E1 -20527.299,E2 -20527.299} C_VEL
LIN {X 0,Y 221.06,Z 335.449,A -85,B 0,C 180,E1 -20530.996,E2 -20530.996} C_VEL
LIN {X 0,Y 220.967,Z 335.434,A -85,B 0,C 180,E1 -20536.633,E2 -20536.633} C_VEL
LIN {X 0,Y 220.85,Z 335.473,A -85,B 0,C 180,E1 -20540.49,E2 -20540.49} C_VEL
LIN {X 0,Y 220.845,Z 335.448,A -85,B 0,C 180,E1 -20544.437,E2 -20544.437} C_VEL
LIN {X 0,Y 220.804,Z 335.48,A -85,B 0,C 180,E1 -20548.517,E2 -20548.517} C_VEL
LIN {X 0,Y 220.812,Z 335.469,A -85,B 0,C 180,E1 -20552.756,E2 -20552.756} C_VEL
LIN {X 0,Y 220.821,Z 335.463,A -85,B 0,C 180,E1 -20557.215,E2 -20557.215} C_VEL
LIN {X 0,Y 219.186,Z 335.679,A -85,B 0,C 180,E1 -20559.225,E2 -20559.225} C_VEL
LIN {X 0,Y 214.585,Z 336.245,A -85,B 0,C 180,E1 -20563.242,E2 -20563.242} C_VEL
LIN {X 0,Y 213.647,Z 336.359,A -85,B 0,C 180,E1 -20565.343,E2 -20565.343} C_VEL
LIN {X 0,Y 213.751,Z 336.448,A -85,B 0,C 180,E1 -20570.428,E2 -20570.428} C_VEL
LIN {X 0,Y 215.274,Z 342.551,A -85,B 0,C 180,E1 -20573.629,E2 -20573.629} C_VEL
LIN {X 0,Y 216.794,Z 346.153,A -85,B 0,C 180,E1 -20574.139,E2 -20574.139} C_VEL
LIN {X 0,Y 224.809,Z 364.465,A -85,B 0,C 180,E1 -20576.063,E2 -20576.063} C_VEL
LIN {X 0,Y 230.28,Z 378.939,A -85,B 0,C 180,E1 -20577.366,E2 -20577.366} C_VEL
LIN {X 0,Y 232.251,Z 393.094,A -85,B 0,C 180,E1 -20578.142,E2 -20578.142} C_VEL
LIN {X 0,Y 229.858,Z 449.849,A -85,B 0,C 180,E1 -20579.949,E2 -20579.949} C_VEL
LIN {X 0,Y 229.133,Z 459.526,A -85,B 0,C 180,E1 -20580.433,E2 -20580.433} C_VEL
LIN {X 0,Y 228.058,Z 469.107,A -85,B 0,C 180,E1 -20581.09,E2 -20581.09} C_VEL
LIN {X 0,Y 226.559,Z 479.327,A -85,B 0,C 180,E1 -20582.018,E2 -20582.018} C_VEL
LIN {X 0,Y 224.815,Z 489.97,A -85,B 0,C 180,E1 -20583.296,E2 -20583.296} C_VEL
LIN {X 0,Y 222.798,Z 499.933,A -85,B 0,C 180,E1 -20584.795,E2 -20584.795} C_VEL
LIN {X 0,Y 221.024,Z 508.251,A -85,B 0,C 180,E1 -20586.331,E2 -20586.331} C_VEL
LIN {X 0,Y 219.066,Z 517.132,A -85,B 0,C 180,E1 -20588.351,E2 -20588.351} C_VEL
LIN {X 0,Y 217.533,Z 523.844,A -85,B 0,C 180,E1 -20590.17,E2 -20590.17} C_VEL
LIN {X 0,Y 215.794,Z 530.858,A -85,B 0,C 180,E1 -20592.467,E2 -20592.467} C_VEL
LIN {X 0,Y 214.251,Z 536.708,A -85,B 0,C 180,E1 -20594.786,E2 -20594.786} C_VEL
LIN {X 0,Y 212.974,Z 542.378,A -85,B 0,C 180,E1 -20597.614,E2 -20597.614} C_VEL
LIN {X 0,Y 212.122,Z 546.831,A -85,B 0,C 180,E1 -20600.464,E2 -20600.464} C_VEL
LIN {X 0,Y 211.727,Z 549.159,A -85,B 0,C 180,E1 -20602.37,E2 -20602.37} C_VEL
LIN {X 0,Y 211.353,Z 552.554,A -85,B 0,C 180,E1 -20606.187,E2 -20606.187} C_VEL
LIN {X 0,Y 211.432,Z 554.137,A -85,B 0,C 180,E1 -20610,E2 -20610} C_VEL
LIN {X 0,Y 211.372,Z 554.438,A -85,B 0,C 180,E1 -20611.905,E2 -20611.905} C_VEL
LIN {X 0,Y 211.563,Z 553.628,A -85,B 0,C 180,E1 -20615.719,E2 -20615.719} C_VEL
LIN {X 0,Y 211.812,Z 552.648,A -85,B 0,C 180,E1 -20617.627,E2 -20617.627} C_VEL
LIN {X 0,Y 212.805,Z 549.494,A -85,B 0,C 180,E1 -20621.429,E2 -20621.429} C_VEL
LIN {X 0,Y 214.063,Z 545.953,A -85,B 0,C 180,E1 -20624.255,E2 -20624.255} C_VEL
LIN {X 0,Y 215.84,Z 541.321,A -85,B 0,C 180,E1 -20627.041,E2 -20627.041} C_VEL
LIN {X 0,Y 218.155,Z 535.453,A -85,B 0,C 180,E1 -20629.771,E2 -20629.771} C_VEL
LIN {X 0,Y 220.859,Z 527.543,A -85,B 0,C 180,E1 -20632.66,E2 -20632.66} C_VEL
LIN {X 0,Y 223.266,Z 520.769,A -85,B 0,C 180,E1 -20634.651,E2 -20634.651} C_VEL
LIN {X 0,Y 225.9,Z 512.833,A -85,B 0,C 180,E1 -20636.565,E2 -20636.565} C_VEL
LIN {X 0,Y 228.479,Z 504.435,A -85,B 0,C 180,E1 -20638.225,E2 -20638.225} C_VEL
LIN {X 0,Y 231.305,Z 494.197,A -85,B 0,C 180,E1 -20639.837,E2 -20639.837} C_VEL
LIN {X 0,Y 233.473,Z 484.871,A -85,B 0,C 180,E1 -20641.03,E2 -20641.03} C_VEL
LIN {X 0,Y 235.56,Z 474.145,A -85,B 0,C 180,E1 -20642.103,E2 -20642.103} C_VEL
LIN {X 0,Y 237.296,Z 463.308,A -85,B 0,C 180,E1 -20642.908,E2 -20642.908} C_VEL
LIN {X 0,Y 238.555,Z 452.772,A -85,B 0,C 180,E1 -20643.468,E2 -20643.468} C_VEL
LIN {X 0,Y 239.58,Z 435.4,A -85,B 0,C 180,E1 -20644.079,E2 -20644.079} C_VEL
LIN {X 0,Y 241.613,Z 395.424,A -85,B 0,C 180,E1 -20645.287,E2 -20645.287} C_VEL
LIN {X 0,Y 240.711,Z 389.452,A -85,B 0,C 180,E1 -20645.714,E2 -20645.714} C_VEL
LIN {X 0,Y 235.427,Z 376.706,A -85,B 0,C 180,E1 -20647.385,E2 -20647.385} C_VEL
LIN {X 0,Y 229.568,Z 364.923,A -85,B 0,C 180,E1 -20649.29,E2 -20649.29} C_VEL
LIN {X 0,Y 224.216,Z 355.594,A -85,B 0,C 180,E1 -20651.133,E2 -20651.133} C_VEL
LIN {X 0,Y 220.335,Z 349.425,A -85,B 0,C 180,E1 -20652.566,E2 -20652.566} C_VEL
LIN {X 0,Y 218.197,Z 346.073,A -85,B 0,C 180,E1 -20653.393,E2 -20653.393} C_VEL
LIN {X 0,Y 215.528,Z 341.939,A -85,B 0,C 180,E1 -20654.497,E2 -20654.497} C_VEL
LIN {X 0,Y 214.905,Z 340.285,A -85,B 0,C 180,E1 -20655.325,E2 -20655.325} C_VEL
LIN {X 0,Y 213.729,Z 336.395,A -85,B 0,C 180,E1 -20658.291,E2 -20658.291} C_VEL
LIN {X 0,Y 213.729,Z 336.356,A -85,B 0,C 180,E1 -20662.109,E2 -20662.109} C_VEL
LIN {X 0,Y 213.756,Z 336.354,A -85,B 0,C 180,E1 -20666.018,E2 -20666.018} C_VEL
LIN {X 0,Y 213.78,Z 336.356,A -85,B 0,C 180,E1 -20670.455,E2 -20670.455} C_VEL
LIN {X 0,Y 213.802,Z 336.354,A -85,B 0,C 180,E1 -20674.702,E2 -20674.702} C_VEL
LIN {X 0,Y 213.814,Z 336.35,A -85,B 0,C 180,E1 -20678.804,E2 -20678.804} C_VEL
LIN {X 0,Y 213.944,Z 336.326,A -85,B 0,C 180,E1 -20682.804,E2 -20682.804} C_VEL
LIN {X 0,Y 213.981,Z 336.315,A -85,B 0,C 180,E1 -20686.709,E2 -20686.709} C_VEL
LIN {X 0,Y 214.197,Z 336.289,A -85,B 0,C 180,E1 -20690.558,E2 -20690.558} C_VEL
LIN {X 0,Y 214.113,Z 336.309,A -85,B 0,C 180,E1 -20694.349,E2 -20694.349} C_VEL
LIN {X 0,Y 214.448,Z 336.273,A -85,B 0,C 180,E1 -20698.122,E2 -20698.122} C_VEL
LIN {X 0,Y 214.552,Z 336.247,A -85,B 0,C 180,E1 -20700,E2 -20700} C_VEL
LIN {X 0,Y 214.448,Z 336.267,A -85,B 0,C 180,E1 -20701.879,E2 -20701.879} C_VEL
LIN {X 0,Y 214.25,Z 336.294,A -85,B 0,C 180,E1 -20707.54,E2 -20707.54} C_VEL
LIN {X 0,Y 214.028,Z 336.322,A -85,B 0,C 180,E1 -20711.363,E2 -20711.363} C_VEL
LIN {X 0,Y 213.935,Z 336.331,A -85,B 0,C 180,E1 -20715.237,E2 -20715.237} C_VEL
LIN {X 0,Y 213.837,Z 336.342,A -85,B 0,C 180,E1 -20719.188,E2 -20719.188} C_VEL
LIN {X 0,Y 213.851,Z 336.5,A -85,B 0,C 180,E1 -20720.187,E2 -20720.187} C_VEL
LIN {X 0,Y 214.232,Z 337.956,A -85,B 0,C 180,E1 -20721.091,E2 -20721.091} C_VEL
LIN {X 0,Y 216.964,Z 341.923,A -85,B 0,C 180,E1 -20722.247,E2 -20722.247} C_VEL
LIN {X 0,Y 222,Z 349.268,A -85,B 0,C 180,E1 -20724.166,E2 -20724.166} C_VEL
LIN {X 0,Y 227.009,Z 357.33,A -85,B 0,C 180,E1 -20725.946,E2 -20725.946} C_VEL
LIN {X 0,Y 233.39,Z 368.888,A -85,B 0,C 180,E1 -20728.056,E2 -20728.056} C_VEL
LIN {X 0,Y 239.192,Z 381.237,A -85,B 0,C 180,E1 -20729.874,E2 -20729.874} C_VEL
LIN {X 0,Y 242.073,Z 388.381,A -85,B 0,C 180,E1 -20730.767,E2 -20730.767} C_VEL
LIN {X 0,Y 238.939,Z 444.066,A -85,B 0,C 180,E1 -20732.457,E2 -20732.457} C_VEL
LIN {X 0,Y 237.959,Z 454.035,A -85,B 0,C 180,E1 -20732.921,E2 -20732.921} C_VEL
LIN {X 0,Y 236.68,Z 463.75,A -85,B 0,C 180,E1 -20733.562,E2 -20733.562} C_VEL
LIN {X 0,Y 234.988,Z 473.802,A -85,B 0,C 180,E1 -20734.443,E2 -20734.443} C_VEL
LIN {X 0,Y 233.069,Z 483.231,A -85,B 0,C 180,E1 -20735.496,E2 -20735.496} C_VEL
LIN {X 0,Y 230.665,Z 493.135,A -85,B 0,C 180,E1 -20736.89,E2 -20736.89} C_VEL
LIN {X 0,Y 227.962,Z 502.845,A -85,B 0,C 180,E1 -20738.607,E2 -20738.607} C_VEL
LIN {X 0,Y 225.204,Z 511.567,A -85,B 0,C 180,E1 -20740.512,E2 -20740.512} C_VEL
LIN {X 0,Y 222.347,Z 519.683,A -85,B 0,C 180,E1 -20742.702,E2 -20742.702} C_VEL
LIN {X 0,Y 220.292,Z 525.433,A -85,B 0,C 180,E1 -20744.577,E2 -20744.577} C_VEL
LIN {X 0,Y 217.703,Z 532.17,A -85,B 0,C 180,E1 -20747.318,E2 -20747.318} C_VEL
LIN {X 0,Y 216.033,Z 536.413,A -85,B 0,C 180,E1 -20749.41,E2 -20749.41} C_VEL
LIN {X 0,Y 214.034,Z 541.517,A -85,B 0,C 180,E1 -20752.758,E2 -20752.758} C_VEL
LIN {X 0,Y 212.741,Z 544.764,A -85,B 0,C 180,E1 -20755.679,E2 -20755.679} C_VEL
LIN {X 0,Y 211.991,Z 546.645,A -85,B 0,C 180,E1 -20757.965,E2 -20757.965} C_VEL
LIN {X 0,Y 211.491,Z 547.717,A -85,B 0,C 180,E1 -20760.102,E2 -20760.102} C_VEL
LIN {X 0,Y 210.994,Z 548.58,A -85,B 0,C 180,E1 -20764.073,E2 -20764.073} C_VEL
LIN {X 0,Y 210.901,Z 548.18,A -85,B 0,C 180,E1 -20766.429,E2 -20766.429} C_VEL
LIN {X 0,Y 211.055,Z 547.172,A -85,B 0,C 180,E1 -20768.81,E2 -20768.81} C_VEL
LIN {X 0,Y 211.248,Z 546.107,A -85,B 0,C 180,E1 -20770.568,E2 -20770.568} C_VEL
LIN {X 0,Y 211.601,Z 544.354,A -85,B 0,C 180,E1 -20772.607,E2 -20772.607} C_VEL
LIN {X 0,Y 212.352,Z 540.822,A -85,B 0,C 180,E1 -20775.628,E2 -20775.628} C_VEL
LIN {X 0,Y 213.343,Z 536.133,A -85,B 0,C 180,E1 -20778.6,E2 -20778.6} C_VEL
LIN {X 0,Y 214.786,Z 530.092,A -85,B 0,C 180,E1 -20781.533,E2 -20781.533} C_VEL
LIN {X 0,Y 216.693,Z 522.412,A -85,B 0,C 180,E1 -20784.417,E2 -20784.417} C_VEL
LIN {X 0,Y 218.506,Z 515.086,A -85,B 0,C 180,E1 -20786.645,E2 -20786.645} C_VEL
LIN {X 0,Y 220.355,Z 507.177,A -85,B 0,C 180,E1 -20788.63,E2 -20788.63} C_VEL
LIN {X 0,Y 222.378,Z 498.275,A -85,B 0,C 180,E1 -20790.453,E2 -20790.453} C_VEL
LIN {X 0,Y 224.379,Z 488.299,A -85,B 0,C 180,E1 -20792.107,E2 -20792.107} C_VEL
LIN {X 0,Y 225.975,Z 479.137,A -85,B 0,C 180,E1 -20793.344,E2 -20793.344} C_VEL
LIN {X 0,Y 227.511,Z 468.984,A -85,B 0,C 180,E1 -20794.429,E2 -20794.429} C_VEL
LIN {X 0,Y 228.764,Z 457.839,A -85,B 0,C 180,E1 -20795.339,E2 -20795.339} C_VEL
LIN {X 0,Y 229.809,Z 446.625,A -85,B 0,C 180,E1 -20795.969,E2 -20795.969} C_VEL
LIN {X 0,Y 230.763,Z 428.551,A -85,B 0,C 180,E1 -20796.597,E2 -20796.597} C_VEL
LIN {X 0,Y 232.627,Z 381.317,A -85,B 0,C 180,E1 -20798.064,E2 -20798.064} C_VEL
LIN {X 0,Y 229.166,Z 371.272,A -85,B 0,C 180,E1 -20798.892,E2 -20798.892} C_VEL
LIN {X 0,Y 220.711,Z 350.931,A -85,B 0,C 180,E1 -20800.878,E2 -20800.878} C_VEL
LIN {X 0,Y 214.4,Z 338.014,A -85,B 0,C 180,E1 -20802.456,E2 -20802.456} C_VEL
LIN {X 0,Y 214.001,Z 336.565,A -85,B 0,C 180,E1 -20803.073,E2 -20803.073} C_VEL
LIN {X 0,Y 213.935,Z 336.333,A -85,B 0,C 180,E1 -20807.695,E2 -20807.695} C_VEL
LIN {X 0,Y 213.813,Z 336.338,A -85,B 0,C 180,E1 -20813.231,E2 -20813.231} C_VEL
LIN {X 0,Y 213.831,Z 336.335,A -85,B 0,C 180,E1 -20817.45,E2 -20817.45} C_VEL
LIN {X 0,Y 213.772,Z 336.355,A -85,B 0,C 180,E1 -20821.737,E2 -20821.737} C_VEL
LIN {X 0,Y 213.755,Z 336.35,A -85,B 0,C 180,E1 -20826.286,E2 -20826.286} C_VEL
LIN {X 0,Y 213.719,Z 336.337,A -85,B 0,C 180,E1 -20831.124,E2 -20831.124} C_VEL
LIN {X 0,Y 213.711,Z 336.351,A -85,B 0,C 180,E1 -20833.678,E2 -20833.678} C_VEL
LIN {X 0,Y 213.71,Z 336.365,A -85,B 0,C 180,E1 -20836.343,E2 -20836.343} C_VEL
LIN {X 0,Y 213.72,Z 336.334,A -85,B 0,C 180,E1 -20839.143,E2 -20839.143} C_VEL
LIN {X 0,Y 213.746,Z 336.352,A -85,B 0,C 180,E1 -20843.712,E2 -20843.712} C_VEL
LIN {X 0,Y 213.761,Z 336.335,A -85,B 0,C 180,E1 -20848.261,E2 -20848.261} C_VEL
LIN {X 0,Y 213.791,Z 336.323,A -85,B 0,C 180,E1 -20852.598,E2 -20852.598} C_VEL
LIN {X 0,Y 213.814,Z 336.348,A -85,B 0,C 180,E1 -20856.978,E2 -20856.978} C_VEL
LIN {X 0,Y 213.888,Z 336.291,A -85,B 0,C 180,E1 -20862.344,E2 -20862.344} C_VEL
LIN {X 0,Y 213.945,Z 336.33,A -85,B 0,C 180,E1 -20866.706,E2 -20866.706} C_VEL
LIN {X 0,Y 214.136,Z 336.292,A -85,B 0,C 180,E1 -20870.555,E2 -20870.555} C_VEL
LIN {X 0,Y 214.077,Z 336.271,A -85,B 0,C 180,E1 -20874.347,E2 -20874.347} C_VEL
LIN {X 0,Y 214.407,Z 336.271,A -85,B 0,C 180,E1 -20878.121,E2 -20878.121} C_VEL
LIN {X 0,Y 214.516,Z 336.262,A -85,B 0,C 180,E1 -20880,E2 -20880} C_VEL
LIN {X 0,Y 214.408,Z 336.26,A -85,B 0,C 180,E1 -20881.878,E2 -20881.878} C_VEL
LIN {X 0,Y 214.191,Z 336.285,A -85,B 0,C 180,E1 -20887.541,E2 -20887.541} C_VEL
LIN {X 0,Y 213.99,Z 336.325,A -85,B 0,C 180,E1 -20891.364,E2 -20891.364} C_VEL
LIN {X 0,Y 213.868,Z 336.308,A -85,B 0,C 180,E1 -20895.241,E2 -20895.241} C_VEL
LIN {X 0,Y 213.792,Z 336.353,A -85,B 0,C 180,E1 -20899.191,E2 -20899.191} C_VEL
LIN {X 0,Y 213.794,Z 336.326,A -85,B 0,C 180,E1 -20903.232,E2 -20903.232} C_VEL
LIN {X 0,Y 213.788,Z 336.355,A -85,B 0,C 180,E1 -20907.427,E2 -20907.427} C_VEL
LIN {X 0,Y 213.759,Z 336.338,A -85,B 0,C 180,E1 -20911.738,E2 -20911.738} C_VEL
LIN {X 0,Y 213.74,Z 336.349,A -85,B 0,C 180,E1 -20916.288,E2 -20916.288} C_VEL
LIN {X 0,Y 213.694,Z 336.36,A -85,B 0,C 180,E1 -20921.129,E2 -20921.129} C_VEL
LIN {X 0,Y 213.647,Z 336.359,A -85,B 0,C 180,E1 -20925.343,E2 -20925.343} C_VEL
LIN {X 0,Y 212.973,Z 336.455,A -85,B 0,C 180,E1 -20926.417,E2 -20926.417} C_VEL
LIN {X 0,Y 210.133,Z 336.811,A -85,B 0,C 180,E1 -20928.113,E2 -20928.113} C_VEL
LIN {X 0,Y 207.532,Z 337.956,A -85,B 0,C 180,E1 -20929.794,E2 -20929.794} C_VEL
LIN {X 0,Y 207.203,Z 339.383,A -85,B 0,C 180,E1 -20930.808,E2 -20930.808} C_VEL
LIN {X 0,Y 208.089,Z 342.695,A -85,B 0,C 180,E1 -20932.468,E2 -20932.468} C_VEL
LIN {X 0,Y 215.064,Z 358.009,A -85,B 0,C 180,E1 -20934.338,E2 -20934.338} C_VEL
LIN {X 0,Y 221.89,Z 374.862,A -85,B 0,C 180,E1 -20936.04,E2 -20936.04} C_VEL
LIN {X 0,Y 224.289,Z 381.583,A -85,B 0,C 180,E1 -20936.641,E2 -20936.641} C_VEL
LIN {X 0,Y 225.978,Z 394.31,A -85,B 0,C 180,E1 -20937.357,E2 -20937.357} C_VEL
LIN {X 0,Y 223.499,Z 449.403,A -85,B 0,C 180,E1 -20939.143,E2 -20939.143} C_VEL
LIN {X 0,Y 222.776,Z 459.038,A -85,B 0,C 180,E1 -20939.63,E2 -20939.63} C_VEL
LIN {X 0,Y 221.675,Z 468.746,A -85,B 0,C 180,E1 -20940.305,E2 -20940.305} C_VEL
LIN {X 0,Y 219.949,Z 479.957,A -85,B 0,C 180,E1 -20941.361,E2 -20941.361} C_VEL
LIN {X 0,Y 218.483,Z 488.955,A -85,B 0,C 180,E1 -20942.457,E2 -20942.457} C_VEL
LIN {X 0,Y 216.359,Z 499.078,A -85,B 0,C 180,E1 -20943.99,E2 -20943.99} C_VEL
LIN {X 0,Y 214.241,Z 508.554,A -85,B 0,C 180,E1 -20945.792,E2 -20945.792} C_VEL
LIN {X 0,Y 212.357,Z 516.851,A -85,B 0,C 180,E1 -20947.732,E2 -20947.732} C_VEL
LIN {X 0,Y 210.435,Z 524.782,A -85,B 0,C 180,E1 -20949.994,E2 -20949.994} C_VEL
LIN {X 0,Y 208.658,Z 531.586,A -85,B 0,C 180,E1 -20952.354,E2 -20952.354} C_VEL
LIN {X 0,Y 207.394,Z 536.296,A -85,B 0,C 180,E1 -20954.27,E2 -20954.27} C_VEL
LIN {X 0,Y 206.007,Z 542.044,A -85,B 0,C 180,E1 -20957.188,E2 -20957.188} C_VEL
LIN {X 0,Y 205.109,Z 546.557,A -85,B 0,C 180,E1 -20960.135,E2 -20960.135} C_VEL
LIN {X 0,Y 204.674,Z 548.885,A -85,B 0,C 180,E1 -20962.105,E2 -20962.105} C_VEL
LIN {X 0,Y 204.252,Z 552.467,A -85,B 0,C 180,E1 -20966.226,E2 -20966.226} C_VEL
LIN {X 0,Y 204.335,Z 554.014,A -85,B 0,C 180,E1 -20970,E2 -20970} C_VEL
LIN {X 0,Y 204.279,Z 554.321,A -85,B 0,C 180,E1 -20971.971,E2 -20971.971} C_VEL
LIN {X 0,Y 204.493,Z 553.599,A -85,B 0,C 180,E1 -20975.918,E2 -20975.918} C_VEL
LIN {X 0,Y 204.748,Z 552.618,A -85,B 0,C 180,E1 -20977.891,E2 -20977.891} C_VEL
LIN {X 0,Y 205.839,Z 549.552,A -85,B 0,C 180,E1 -20981.821,E2 -20981.821} C_VEL
LIN {X 0,Y 207.164,Z 546.065,A -85,B 0,C 180,E1 -20984.74,E2 -20984.74} C_VEL
LIN {X 0,Y 209.075,Z 541.503,A -85,B 0,C 180,E1 -20987.61,E2 -20987.61} C_VEL
LIN {X 0,Y 211.904,Z 534.568,A -85,B 0,C 180,E1 -20990.887,E2 -20990.887} C_VEL
LIN {X 0,Y 214.232,Z 528.227,A -85,B 0,C 180,E1 -20993.286,E2 -20993.286} C_VEL
LIN {X 0,Y 216.868,Z 521.222,A -85,B 0,C 180,E1 -20995.429,E2 -20995.429} C_VEL
LIN {X 0,Y 219.959,Z 512.377,A -85,B 0,C 180,E1 -20997.6,E2 -20997.6} C_VEL
LIN {X 0,Y 222.626,Z 503.91,A -85,B 0,C 180,E1 -20999.295,E2 -20999.295} C_VEL
LIN {X 0,Y 225.224,Z 495.059,A -85,B 0,C 180,E1 -21000.729,E2 -21000.729} C_VEL
LIN {X 0,Y 227.847,Z 484.14,A -85,B 0,C 180,E1 -21002.146,E2 -21002.146} C_VEL
LIN {X 0,Y 229.835,Z 474.446,A -85,B 0,C 180,E1 -21003.133,E2 -21003.133} C_VEL
LIN {X 0,Y 231.731,Z 462.989,A -85,B 0,C 180,E1 -21003.999,E2 -21003.999} C_VEL
LIN {X 0,Y 233.064,Z 452.365,A -85,B 0,C 180,E1 -21004.561,E2 -21004.561} C_VEL
LIN {X 0,Y 234.166,Z 434.49,A -85,B 0,C 180,E1 -21005.197,E2 -21005.197} C_VEL
LIN {X 0,Y 236.186,Z 396.642,A -85,B 0,C 180,E1 -21006.364,E2 -21006.364} C_VEL
LIN {X 0,Y 235.445,Z 392.039,A -85,B 0,C 180,E1 -21006.721,E2 -21006.721} C_VEL
LIN {X 0,Y 230.49,Z 380.076,A -85,B 0,C 180,E1 -21008.372,E2 -21008.372} C_VEL
LIN {X 0,Y 225.062,Z 368.896,A -85,B 0,C 180,E1 -21010.262,E2 -21010.262} C_VEL
LIN {X 0,Y 220.171,Z 360.273,A -85,B 0,C 180,E1 -21012.044,E2 -21012.044} C_VEL
LIN {X 0,Y 216.711,Z 354.653,A -85,B 0,C 180,E1 -21013.386,E2 -21013.386} C_VEL
LIN {X 0,Y 214.593,Z 351.339,A -85,B 0,C 180,E1 -21014.242,E2 -21014.242} C_VEL
LIN {X 0,Y 211.088,Z 346.091,A -85,B 0,C 180,E1 -21015.721,E2 -21015.721} C_VEL
LIN {X 0,Y 207.93,Z 341.251,A -85,B 0,C 180,E1 -21017.305,E2 -21017.305} C_VEL
LIN {X 0,Y 206.772,Z 337.96,A -85,B 0,C 180,E1 -21019.775,E2 -21019.775} C_VEL
LIN {X 0,Y 206.669,Z 337.251,A -85,B 0,C 180,E1 -21020.689,E2 -21020.689} C_VEL
LIN {X 0,Y 206.698,Z 337.229,A -85,B 0,C 180,E1 -21024.689,E2 -21024.689} C_VEL
LIN {X 0,Y 206.713,Z 337.227,A -85,B 0,C 180,E1 -21029.338,E2 -21029.338} C_VEL
LIN {X 0,Y 206.733,Z 337.226,A -85,B 0,C 180,E1 -21033.773,E2 -21033.773} C_VEL
LIN {X 0,Y 206.758,Z 337.221,A -85,B 0,C 180,E1 -21038.044,E2 -21038.044} C_VEL
LIN {X 0,Y 206.874,Z 337.202,A -85,B 0,C 180,E1 -21042.197,E2 -21042.197} C_VEL
LIN {X 0,Y 206.915,Z 337.195,A -85,B 0,C 180,E1 -21046.246,E2 -21046.246} C_VEL
LIN {X 0,Y 207.133,Z 337.17,A -85,B 0,C 180,E1 -21050.233,E2 -21050.233} C_VEL
LIN {X 0,Y 207.076,Z 337.187,A -85,B 0,C 180,E1 -21054.157,E2 -21054.157} C_VEL
LIN {X 0,Y 207.384,Z 337.152,A -85,B 0,C 180,E1 -21058.058,E2 -21058.058} C_VEL
LIN {X 0,Y 207.517,Z 337.123,A -85,B 0,C 180,E1 -21060,E2 -21060} C_VEL
LIN {X 0,Y 207.384,Z 337.147,A -85,B 0,C 180,E1 -21061.943,E2 -21061.943} C_VEL
LIN {X 0,Y 207.19,Z 337.17,A -85,B 0,C 180,E1 -21067.799,E2 -21067.799} C_VEL
LIN {X 0,Y 206.947,Z 337.2,A -85,B 0,C 180,E1 -21071.758,E2 -21071.758} C_VEL
LIN {X 0,Y 206.868,Z 337.209,A -85,B 0,C 180,E1 -21075.771,E2 -21075.771} C_VEL
LIN {X 0,Y 206.893,Z 337.417,A -85,B 0,C 180,E1 -21078.09,E2 -21078.09} C_VEL
LIN {X 0,Y 207.092,Z 338.454,A -85,B 0,C 180,E1 -21078.526,E2 -21078.526} C_VEL
LIN {X 0,Y 208.506,Z 341.032,A -85,B 0,C 180,E1 -21079.262,E2 -21079.262} C_VEL
LIN {X 0,Y 210.756,Z 343.296,A -85,B 0,C 180,E1 -21080.242,E2 -21080.242} C_VEL
LIN {X 0,Y 214.034,Z 348.005,A -85,B 0,C 180,E1 -21081.639,E2 -21081.639} C_VEL
LIN {X 0,Y 219.066,Z 355.737,A -85,B 0,C 180,E1 -21083.642,E2 -21083.642} C_VEL
LIN {X 0,Y 223.703,Z 363.464,A -85,B 0,C 180,E1 -21085.359,E2 -21085.359} C_VEL
LIN {X 0,Y 229.307,Z 373.932,A -85,B 0,C 180,E1 -21087.308,E2 -21087.308} C_VEL
LIN {X 0,Y 234.724,Z 385.73,A -85,B 0,C 180,E1 -21089.094,E2 -21089.094} C_VEL
LIN {X 0,Y 236.546,Z 390.293,A -85,B 0,C 180,E1 -21089.689,E2 -21089.689} C_VEL
LIN {X 0,Y 233.458,Z 443.855,A -85,B 0,C 180,E1 -21091.359,E2 -21091.359} C_VEL
LIN {X 0,Y 232.451,Z 453.768,A -85,B 0,C 180,E1 -21091.819,E2 -21091.819} C_VEL
